# B&R Automation Studio project ControlPLC_DataDistribution (part 7)

#### vfValveBasic.st
```iecst
FUNCTION_BLOCK vfValveBasic

	pCommandWriteBack ACCESS (Inputs.adrCommands);

	IF NOT (Inputs.parameters.enabled) THEN
		internal.valveState	:= vfVALVE_BASIC_STOP;
	ELSIF(Inputs.commands.stop = TRUE) THEN
		pCommandWriteBack.stop := FALSE;
		internal.valveState	:= vfVALVE_BASIC_STOP;
	END_IF

	CASE internal.valveState OF

		vfVALVE_BASIC_WAIT_FOR_COMMANDS:

			Outputs.status.fbState := 'WAITING FOR COMMANDS';

			Outputs.status.readyForCommand := TRUE;

			IF (Inputs.commands.cycle = TRUE) THEN

				pCommandWriteBack.cycle := FALSE;

				internal.valveState	:= vfVALVE_BASIC_CYCLE_OPEN;

			ELSIF (Inputs.commands.open = TRUE) THEN

				pCommandWriteBack.open := FALSE;

				IF NOT Outputs.status.opened THEN

					internal.valveTimeOutTimer.IN := TRUE;

					internal.valveState	:= vfVALVE_BASIC_OPEN;
				END_IF

			ELSIF (Inputs.commands.close = TRUE)THEN

				pCommandWriteBack.close := FALSE;

				IF NOT Outputs.status.closed THEN

					internal.valveTimeOutTimer.IN := TRUE;

					internal.valveState	:= vfVALVE_BASIC_CLOSE;;
				END_IF

			END_IF

		vfVALVE_BASIC_CYCLE_OPEN:

			Outputs.status.fbState := 'CYCLE OPEN';
			Outputs.OpenValveSignal := TRUE; //cmd
			Outputs.CloseValveSignal := FALSE;//cmd
			Outputs.status.cycling	:= TRUE;//status
			Outputs.status.doOpen 	:= TRUE;//status
			Outputs.status.doClose	:= FALSE;//status

			internal.valveCycleTimer.PT	:= Inputs.parameters.cycleTime;
			internal.valveCycleTimer.IN	:= TRUE;
			internal.valveTimeOutTimer.IN := TRUE;

			//once its opened stop monitoring for timeout error
			IF Outputs.status.opened THEN
				internal.valveTimeOutTimer.IN := FALSE;

			//didnt open after allowed time
			ELSIF internal.valveTimeOutTimer.Q 	THEN
				internal.valveTimeOutTimer.IN := FALSE;
				internal.valveState := vfVALVE_BASIC_ERROR;

			END_IF

			//cycled open long enough
			IF (internal.valveCycleTimer.Q = TRUE) AND Outputs.status.opened THEN
				internal.valveCycleTimer.IN	:= FALSE;
				Outputs.CloseValveSignal := TRUE;
				Outputs.OpenValveSignal := FALSE;
				Outputs.status.doOpen := FALSE;
				Outputs.status.doClose := TRUE;

				//reset timeout timer
				internal.valveTimeOutTimer.IN := FALSE;
				internal.valveState				:= vfVALVE_BASIC_CYCLE_CLOSE;

			END_IF

		vfVALVE_BASIC_CYCLE_CLOSE:

			Outputs.status.fbState := 'CYCLE CLOSE';

			IF Outputs.status.closed THEN
				Outputs.status.cycling := FALSE;
				internal.valveTimeOutTimer.IN := FALSE;
				internal.valveState				:= vfVALVE_BASIC_WAIT_FOR_COMMANDS;

			ELSIF internal.valveTimeOutTimer.Q THEN
				internal.valveTimeOutTimer.IN := FALSE;
				internal.valveState := vfVALVE_BASIC_ERROR;

			END_IF

		vfVALVE_BASIC_OPEN:

			Outputs.status.fbState := 'OPENING';

			//open valve
			Outputs.OpenValveSignal := TRUE;
			Outputs.CloseValveSignal := FALSE;

			//update valve output status
			Outputs.status.doOpen 					:= TRUE;
			Outputs.status.doClose					:= FALSE;

			IF Outputs.status.opened THEN

				//reset timeout timer
				internal.valveTimeOutTimer.IN := FALSE;
				internal.valveState				:= vfVALVE_BASIC_WAIT_FOR_COMMANDS;

			ELSIF internal.valveTimeOutTimer.Q 	THEN

				internal.valveState := vfVALVE_BASIC_ERROR;

			END_IF

		vfVALVE_BASIC_CLOSE:

			Outputs.status.fbState := 'CLOSING';

			Outputs.OpenValveSignal := FALSE;
			Outputs.CloseValveSignal := TRUE;

			//update valve output status
			Outputs.status.doOpen 					:= FALSE;
			Outputs.status.doClose 				:= TRUE;

			IF Outputs.status.closed THEN

				//reset timeout timer
				internal.valveTimeOutTimer.IN := FALSE;
				internal.valveState				:= vfVALVE_BASIC_WAIT_FOR_COMMANDS;

			ELSIF internal.valveTimeOutTimer.Q 	THEN

				internal.valveState := vfVALVE_BASIC_ERROR;

			END_IF

		vfVALVE_BASIC_STOP:

			Outputs.status.fbState := 'STOPPING';

			Outputs.OpenValveSignal := FALSE;
			Outputs.CloseValveSignal := FALSE;

			//reset timeout timer
			internal.valveTimeOutTimer.IN := FALSE;
			internal.valveCycleTimer.IN		:= FALSE;

			//update valve output status
			Outputs.status.cycling					:= FALSE;
			Outputs.status.doOpen 					:= FALSE;
			Outputs.status.doClose 				:= FALSE;
			internal.valveState				:= vfVALVE_BASIC_WAIT_FOR_COMMANDS;

		vfVALVE_BASIC_ERROR:

			Outputs.status.fbState := 'ERRORED';

			//reset timeout timer
			internal.valveTimeOutTimer.IN := FALSE;

			Outputs.status.error := TRUE;

			IF Inputs.commands.errReset THEN

				Outputs.status.error := FALSE;

				internal.valveState				:= vfVALVE_BASIC_WAIT_FOR_COMMANDS;
			END_IF

	END_CASE

	IF (internal.valveState = vfVALVE_BASIC_ERROR) OR (internal.valveState = vfVALVE_BASIC_WAIT_FOR_COMMANDS) THEN
		Outputs.status.busy := FALSE;
	ELSE
		Outputs.status.busy := TRUE;
	END_IF

	//so nothing gets queued and stuck
	IF internal.valveState <> vfVALVE_BASIC_WAIT_FOR_COMMANDS THEN

		Outputs.status.readyForCommand := FALSE;

		pCommandWriteBack.close := FALSE;
		pCommandWriteBack.open := FALSE;
		pCommandWriteBack.cycle := FALSE;

	END_IF

	IF Inputs.commands.errReset THEN
		Outputs.status.error := FALSE;
	END_IF

	//feedback for position
	IF Inputs.parameters.hasLimitSensors THEN

		Outputs.status.closed := Inputs.closeLimitSensor;
		Outputs.status.opened := Inputs.openLimitSensor;

		Outputs.status.middle := NOT(Inputs.closeLimitSensor OR Inputs.openLimitSensor);

		internal.valveTimeOutTimer.PT := Inputs.parameters.TimeOutValue;
		internal.valveTimeOutTimer();

	ELSE

		internal.actuationDelayTimer.PT := Inputs.parameters.actuationDelay;

		IF Outputs.status.doClose AND NOT internal.oldDoClose THEN
			Outputs.status.opened := FALSE;
			internal.actuationDelayTimer.IN := TRUE;

		ELSIF Outputs.status.doOpen AND NOT internal.oldDoOpen THEN
			Outputs.status.closed := FALSE;
			internal.actuationDelayTimer.IN := TRUE;
		END_IF

		IF internal.actuationDelayTimer.Q THEN
			internal.actuationDelayTimer.IN := FALSE;
			Outputs.status.closed := Outputs.status.doClose;
			Outputs.status.opened := Outputs.status.doOpen;
		END_IF

		internal.actuationDelayTimer();

		//for rising edge
		internal.oldDoOpen := Outputs.status.doOpen;
		internal.oldDoClose := Outputs.status.doClose;

	END_IF

	//init timer for cycle option
	internal.valveCycleTimer();

END_FUNCTION_BLOCK
```

- vfValveBasic_readMe.docx (binary file, 312023 bytes)
### Library Logical/Libraries/VF/VF_PARSER (IEC, version 1.00.0)

#### RevisionNotes.txt
```
****************************************************************************************************
IMPORTANT: Always update the library version number in the library Properties 'Details' tab.
****************************************************************************************************

Version 1.00 - 9/23/19, W. Stebler
----------------------------------
- Original version.
```

#### Types.typ - Exported data types
```iecst
(**)
(*ParseLSF structures*)

TYPE
	vfpLSFCommandType : 	STRUCT
		SelectedBuildLayout : UDINT;
		SelectedPrintNumber : UINT;
		SelectedRack : USINT;
		SelectedLayer : UDINT;
		OptionalStartingTrajectory : UINT;
		NumLasersInRack : USINT;
		OpenLayer : BOOL;
		ParseTrajectory : BOOL;
		CloseLayer : BOOL;
		AbortLayer : BOOL;
		ResetError : BOOL;
	END_STRUCT;
	vfpLSFStatusType : 	STRUCT
		LayerFilename : STRING[255];
		LayerOpen : BOOL;
		CurrentLayer : UDINT;
		FinalTrajectoryNumber : UINT;
		ParsedTrajectoryNumber : UINT;
		ParseTrajectoryComplete : BOOL;
		LayerClosed : BOOL;
		LayerAborted : BOOL;
		Error : BOOL;
		ErrorID : UINT;
		ErrorText : STRING[80];
	END_STRUCT;
	vfpLSFInternalFBType : 	STRUCT
		FileOpen : FileOpen;
		FileReadEx : FileReadEx;
		FileClose : FileClose;
	END_STRUCT;
	vfpLSFParsedDataType : 	STRUCT
		TrajectoryCircularBuffer : ARRAY[1..vfp_LSF_TRAJECTORY_FIFO_SIZE]OF vfpLSFBufferElementType;
		FIFOCount : USINT := 0;
		FIFOHeadIndex : USINT := 1;
		FIFOTailIndex : USINT := 1;
	END_STRUCT;
	vfpLSFBufferElementType : 	STRUCT
		TrajectoryNumber : UINT;
		LaserTrajectoryInfo : ARRAY[1..vfp_LSF_NUM_LASERS_PER_SYSTEM]OF vfpLSFLaserTrajectoryInfoType;
		ExitCode : UINT;
	END_STRUCT;
	vfpLSFLaserTrajectoryInfoType : 	STRUCT
		PowerSetpointPercent : REAL;
		NumStateValues : UINT;
		StateValue32Bit : ARRAY[1..vfp_LSF_MAX_32BIT_VAL_PER_TRAJ]OF UDINT;
	END_STRUCT;
	vfpLSFLocalType : 	STRUCT
		Step : vfpLSFStepsEnum;
		StepTrace : ARRAY[0..99]OF vfpLSFStepsEnum;
		index : UINT;
		FB : vfpLSFInternalFBType;
		ErrorStep : vfpLSFStepsEnum;
		DataBuffer : STRING[vfp_LSF_FILE_READ_BUFFER_SIZE];
		ReadLengthBytes : UDINT;
		TotalBytesRead : UDINT;
		StartingByteAddress : UDINT;
		MaxBytes : UDINT;
		NextByteAddress : UDINT;
		CurrentByteIndex : UDINT;
		ParameterValue : LREAL;
		ParameterValue_UDINT : UDINT;
		ParameterValue_string : STRING[vfp_MAX_CHARS_PER_STRING_VALUE];
		ParsedHeaderLine : BOOL;
		FoundTrajectory : BOOL;
		Status : UINT;
		BuildLayout : UDINT;
		PrintNumber : UINT;
		RackNumber : USINT;
		LayerNumber : UDINT;
		LayerClosed : BOOL;
		LayerAborted : BOOL;
		FinalTrajectoryNumber : UINT;
		TrajectoryNumber : UINT;
		LaserNumber : USINT;
		LastLaserNumber : USINT;
		LaserPowerValueIndex : USINT;
		LaserStateValueIndex : UINT;
		ExpectedNumEvents : UINT;
		FileReadOffset : UDINT;
		LocalFileHandle : UDINT;
		GCodeLineNumber_string : STRING[30];
		BuildLayout_string : STRING[20];
		PrintNumber_string : STRING[20];
		RackNumber_string : STRING[8];
		LayerNumber_string : STRING[8];
		LayerFileName : STRING[255];
		HeaderElement : USINT;
		BuildName : STRING[80];
		BuildPlateFormat : STRING[40];
		Temp_val : UINT;
		Temp_string : STRING[40];
	END_STRUCT;
	vfpLSFStepsEnum :
		(
		vfSTEP_LSF_INITIALIZE,
		vfSTEP_LSF_IDLE,
		vfSTEP_LSF_CREATE_LAYER_FILENAME,
		vfSTEP_LSF_OPEN_FILE,
		vfSTEP_LSF_WAIT_FILE_OPEN,
		vfSTEP_LSF_AWAIT_COMMAND,
		vfSTEP_LSF_READ_FILE_DATA,
		vfSTEP_LSF_WAIT_READ_DONE,
		vfSTEP_LSF_PARSE_FILE_HDR,
		vfSTEP_LSF_FIND_TRAJECTORY_HDR,
		vfSTEP_LSF_PARSE_TRAJECTORY_HDR,
		vfSTEP_LSF_PARSE_NUM_EVENTS,
		vfSTEP_LSF_PARSE_LASER_POWERS,
		vfSTEP_LSF_PARSE_LASER_STATES,
		vfSTEP_LSF_SELECT_NEXT_LASER,
		vfSTEP_LSF_TRAJECTORY_PARSE_DONE,
		vfSTEP_LSF_AWAIT_NEXT_COMMAND,
		vfSTEP_LSF_CLOSE_FILE,
		vfSTEP_LSF_WAIT_FILE_CLOSED,
		vfSTEP_LSF_LAYER_CLOSED,
		vfSTEP_LSF_LAYER_ABORTED,
		vfSTEP_LSF_ERROR,
		vfSTEP_LSF_AWAIT_CMD_RESET
		);
END_TYPE

(**)
(*ParseFEF structures*)

TYPE
	vfpFEFCommandType : 	STRUCT
		SelectedBuildLayout : UDINT;
		SelectedPrintNumber : UINT;
		SelectedLayer : UDINT;
		OptionalStartingTrajectory : UINT;
		OpenLayer : BOOL;
		ParseTrajectory : BOOL;
		CloseLayer : BOOL;
		AbortLayer : BOOL;
		ResetError : BOOL;
	END_STRUCT;
	vfpFEFStatusType : 	STRUCT
		LayerFilename_GCode : STRING[255];
		LayerFilename_FixedEvents : STRING[255];
		LayerOpen : BOOL;
		CurrentLayer : UDINT;
		FinalTrajectoryNumber : UINT;
		ParsedTrajectoryNumber : UINT;
		ParseTrajectoryComplete : BOOL;
		LayerClosed : BOOL;
		LayerAborted : BOOL;
		Error : BOOL;
		ErrorID : UINT;
		ErrorText : STRING[80];
	END_STRUCT;
	vfpFEFInternalFBType : 	STRUCT
		FileOpen : FileOpen;
		FileReadEx : FileReadEx;
		FileClose : FileClose;
	END_STRUCT;
	vfpFEFParsedDataType : 	STRUCT
		TrajectoryCircularBuffer : ARRAY[1..vfp_FEF_TRAJECTORY_FIFO_SIZE]OF vfpFEFBufferElementType;
		FIFOCount : USINT := 0;
		FIFOHeadIndex : USINT := 1;
		FIFOTailIndex : USINT := 1;
	END_STRUCT;
	vfpFEFBufferElementType : 	STRUCT
		TrajectoryNumber : UINT;
		ExitCode : UINT;
		MasterAxis : USINT;
		StartPositionMM : REAL;
		EndPositionMM : REAL;
		EventPeriodMM : REAL;
	END_STRUCT;
	vfpFEFLocalType : 	STRUCT
		Step : vfpFEFStepsEnum;
		StepTrace : ARRAY[0..99]OF vfpFEFStepsEnum;
		index : UINT;
		FB : vfpFEFInternalFBType;
		ErrorStep : vfpFEFStepsEnum;
		DataBuffer : STRING[vfp_FEF_FILE_READ_BUFFER_SIZE];
		ReadLengthBytes : UDINT;
		TotalBytesRead : UDINT;
		StartingByteAddress : UDINT;
		MaxBytes : UDINT;
		NextByteAddress : UDINT;
		CurrentByteIndex : UDINT;
		ParameterValue : LREAL;
		ParameterValue_UDINT : UDINT;
		ParameterValue_string : STRING[vfp_MAX_CHARS_PER_STRING_VALUE];
		ParsedHeaderLine : BOOL;
		FoundTrajectory : BOOL;
		Status : UINT;
		BuildLayout : UDINT;
		PrintNumber : UINT;
		LayerNumber : UDINT;
		LayerClosed : BOOL;
		LayerAborted : BOOL;
		FinalTrajectoryNumber : UINT;
		TrajectoryNumber : UINT;
		FileReadOffset : UDINT;
		LocalFileHandle : UDINT;
		MasterAxis : USINT;
		StartPosition : REAL;
		EndPosition : REAL;
		EventPeriod : REAL;
		GCodeLineNumber_string : STRING[30];
		BuildLayout_string : STRING[20];
		PrintNumber_string : STRING[20];
		LayerNumber_string : STRING[8];
		LayerFileName_FixedEvents : STRING[255];
		LayerFileName_GCode : STRING[255];
		HeaderElement : USINT;
		BuildName : STRING[80];
		BuildPlateFormat : STRING[40];
		Temp_val : UINT;
		Temp_string : STRING[40];
	END_STRUCT;
	vfpFEFStepsEnum :
		(
		vfSTEP_FEF_INITIALIZE,
		vfSTEP_FEF_IDLE,
		vfSTEP_FEF_CREATE_LAYER_FILENAME,
		vfSTEP_FEF_OPEN_FILE,
		vfSTEP_FEF_WAIT_FILE_OPEN,
		vfSTEP_FEF_AWAIT_COMMAND,
		vfSTEP_FEF_READ_FILE_DATA,
		vfSTEP_FEF_WAIT_READ_DONE,
		vfSTEP_FEF_PARSE_FILE_HDR,
		vfSTEP_FEF_FIND_TRAJECTORY_HDR,
		vfSTEP_FEF_PARSE_TRAJECTORY_HDR,
		vfSTEP_FEF_PARSE_MASTER_AXIS,
		vfSTEP_FEF_PARSE_START_POSN,
		vfSTEP_FEF_PARSE_END_POSN,
		vfSTEP_FEF_PARSE_EVENT_PERIOD,
		vfSTEP_FEF_TRAJECTORY_PARSE_DONE,
		vfSTEP_FEF_AWAIT_NEXT_COMMAND,
		vfSTEP_FEF_CLOSE_FILE,
		vfSTEP_FEF_WAIT_FILE_CLOSED,
		vfSTEP_FEF_LAYER_CLOSED,
		vfSTEP_FEF_LAYER_ABORTED,
		vfSTEP_FEF_ERROR,
		vfSTEP_FEF_AWAIT_CMD_RESET
		);
END_TYPE

(**)
(*SMRFile structures*)

TYPE
	VfSMRFileInternalType : 	STRUCT
		Step : VfSMRFileStepsEnum;
		StepTrace : ARRAY[0..99]OF VfSMRFileStepsEnum;
		ErrorStep : VfSMRFileStepsEnum;
		FB : VfSMRFileInternalFBType;
		index : UINT;
	END_STRUCT;
	VfSMRFileInternalFBType : 	STRUCT
		FileCopy1 : FileCopy;
		FileCopy2 : FileCopy;
		FileCopy3 : FileCopy;
	END_STRUCT;
	VfSMRFileStepsEnum :
		(
		vfSMR_FILE_STEP_IDLE,
		vfSMR_FILE_STEP_COPY_TO_SMR1,
		vfSMR_FILE_STEP_COPY_TO_SMR2,
		vfSMR_FILE_STEP_COPY_TO_SMR3,
		vfSMR_FILE_STEP_COPY_TO_SMR4,
		vfSMR_FILE_STEP_COPY_TO_PTR1,
		vfSMR_FILE_STEP_COPY_TO_PTR2,
		vfSMR_FILE_STEP_COPY_TO_LCR1,
		vfSMR_FILE_STEP_COPY_TO_LCR2,
		vfSMR_FILE_STEP_DONE,
		vfSMR_FILE_STEP_DISCONNECT1,
		vfSMR_FILE_STEP_DISCONNECT2,
		vfSMR_FILE_STEP_ERROR,
		vfSMR_FILE_STEP_ERROR_RESET
		);
END_TYPE

(**)
(*SMRConnect structures*)

TYPE
	VfSMRConnectInternalType : 	STRUCT
		Step : VfSMRConnectStepsEnum;
		StepTrace : ARRAY[0..99]OF VfSMRConnectStepsEnum;
		ErrorStep : VfSMRConnectStepsEnum;
		FB : VfSMRConnectInternalFBType;
		LocalFileHandle : UDINT;
		index : UINT;
	END_STRUCT;
	VfSMRConnectInternalFBType : 	STRUCT
		DevLinkRemote : DevLink;
		DevLinkLocalSMR : DevLink;
		DevLinkLocalPTR : DevLink;
		DevLinkLocalLCR : DevLink;
		DevUnlinkRemote : DevUnlink;
		DevUnlinkLocalSMR : DevUnlink;
		DevUnlinkLocalPTR : DevUnlink;
		DevUnlinkLocalLCR : DevUnlink;
	END_STRUCT;
	VfSMRConnectStepsEnum :
		(
		vfSMR_CNCT_STEP_IDLE,
		vfSMR_CNCT_STEP_CONNECT_SMR1,
		vfSMR_CNCT_STEP_CONNECT_SMR2,
		vfSMR_CNCT_STEP_CONNECT_PTR1,
		vfSMR_CNCT_STEP_CONNECT_PTR2,
		vfSMR_CNCT_STEP_CONNECT_LCR1,
		vfSMR_CNCT_STEP_CONNECT_LCR2,
		vfSMR_CNCT_STEP_CONNECT_REMOTE1,
		vfSMR_CNCT_STEP_CONNECT_REMOTE2,
		vfSMR_CNCT_STEP_DONE,
		vfSMR_CNCT_STEP_DISCONNECT1,
		vfSMR_CNCT_STEP_DISCONNECT2,
		vfSMR_CNCT_STEP_ERROR,
		vfSMR_CNCT_STEP_ERROR_RESET
		);
END_TYPE

(**)
(*LCRConnect structures*)

TYPE
	VfLCRConnectInternalType : 	STRUCT
		Step : VfLCRConnectStepsEnum;
		StepTrace : ARRAY[0..99]OF VfLCRConnectStepsEnum;
		ErrorStep : VfLCRConnectStepsEnum;
		FB : VfLCRConnectInternalFBType;
		LocalFileName : STRING[80];
		LocalLCRDriveName : STRING[80];
		LocalFileHandle : UDINT;
		i : UINT;
	END_STRUCT;
	VfLCRConnectInternalFBType : 	STRUCT
		DevLinkLocalLCR : DevLink;
		DevUnlinkLocalLCR : DevUnlink;
	END_STRUCT;
	VfLCRConnectStepsEnum :
		(
		vfLCR_CNCT_STEP_IDLE,
		vfLCR_CNCT_STEP_CONNECT_LCR1,
		vfLCR_CNCT_STEP_CONNECT_LCR2,
		vfLCR_CNCT_STEP_DONE,
		vfLCR_CNCT_STEP_DISCONNECT1,
		vfLCR_CNCT_STEP_DISCONNECT2,
		vfLCR_CNCT_STEP_ERROR,
		vfLCR_CNCT_STEP_ERROR_RESET
		);
END_TYPE
```

#### Constants.var - Exported constants
```iecst
(*Shared parser constants*)
VAR CONSTANT
	vfp_MAX_CHARS_PER_STRING_VALUE : UINT := 60; (*Maximum characters allowed for any string value*)
	vfp_MAX_CHARS_PER_NUMERIC_VALUE : UINT := 30; (*Maximum characters allowed for any numeric value (including decimal point, negative sign, delimiter)*)
	fvp_FIRST_TRAJECTORY_NUMBER : UINT := 10; (*Trajectories start at N0010 and increment by 10 (N0010, N0020, N0030,...)*)
	fvp_TRAJECTORY_NUMBER_INCREMENT : USINT := 10;
END_VAR
(*Laser State File (LSF) parser constants*)
VAR CONSTANT
	vfp_LSF_FILE_READ_BUFFER_SIZE : UDINT := 341000; (*> maximum single trajectory (1630 values * 11 bytes * 19 lasers)*)
	vfp_LSF_TRAJECTORY_FIFO_SIZE : USINT := 4;
	vfp_LSF_NUM_LASERS_PER_SYSTEM : UINT := 19;
	vfp_LSF_MAX_32BIT_VAL_PER_TRAJ : UINT := 1630; (*52000 events / 32 bits = 1625 (+ 5 extra for padding)*)
	vfp_LSF_MAX_CHARS_PER_32BIT_VAL : UINT := 11; (*Maximum characters allowed for a laser state event (10 digit value + delimiter) [10 digits required to represent max UDINT value of 4,294,967,295]*)
	vfp_LSF_MAX_CHARS_PER_HEADER : UINT := 300; (*Maximum characters allowed for a single trajectory header information*)
END_VAR
(*Fixed Event File (FEF) parser constants*)
VAR CONSTANT
	vfp_FEF_FILE_READ_BUFFER_SIZE : UDINT := 200;
	vfp_FEF_TRAJECTORY_FIFO_SIZE : USINT := 100;
	vfp_FEF_MASTER_AXIS_X : USINT := 1;
	vfp_FEF_MASTER_AXIS_Y : USINT := 2;
	vfp_FEF_MAX_X_Y_POSN_MM : LREAL := 960.0;
END_VAR
(*Common parser ASCII character codes*)
VAR CONSTANT
	vfp_CHAR_CARRIAGE_RETURN : USINT := 13; (*Carriage Return ASCII char*)
	vfp_CHAR_LINE_FEED : USINT := 10; (*Line Feed ASCII char*)
	vfp_CHAR_SPACE : USINT := 32; (*Space ASCII char*)
	vfp_CHAR_COMMA : USINT := 44; (*',' ASCII char*)
	vfp_CHAR_DECIMAL_POINT : USINT := 46; (*'.' ASCII char*)
	vfp_CHAR_DIGIT_0 : USINT := 48; (*'0' ASCII char*)
	vfp_CHAR_DIGIT_9 : USINT := 57; (*'9' ASCII char*)
	vfp_CHAR_EQUALS : USINT := 61; (*'=' ASCII char*)
	vfp_CHAR_TRAJECTORY_HDR : USINT := 78; (*'N' ASCII char*)
END_VAR
(*Common parser return codes*)
VAR CONSTANT
	vfp_ERR_OK : UINT := 50000;
	vfp_ERR_EOL_REACHED : UINT := 50001;
	vfp_ERR_NO_MORE_LINES : UINT := 50002;
	vfp_ERR_NULL_POINTER : UINT := 50003;
	vfp_ERR_INVALID_PARAMETER : UINT := 50004;
	vfp_ERR_NO_DELIMITER : UINT := 50005;
	vfp_ERR_MISSING_DATA : UINT := 50006;
	vfp_ERR_NON_NUMERICAL : UINT := 50007;
	vfp_ERR_WRONG_NUM_STATES : UINT := 50008;
	vfp_ERR_BAD_HEADER : UINT := 50009;
	vfp_ERR_HEADER_INVALID_NUM_TRAJ : UINT := 50010;
	vfp_ERR_BUFFER_SIZE : UINT := 50040;
	vfp_ERR_FATAL_SYSTEM_ERROR : UINT := 50050;
END_VAR
(**)
```

#### VF_PARSER.fun - Exported functions and function blocks
```iecst
{REDUND_ERROR} FUNCTION GetNextString : UINT (* *) (*$GROUP=User,$CAT=User,$GROUPICON=User.png,$CATICON=User.png*)
	VAR_INPUT
		pAdrData : UDINT;
		pParameter : UDINT;
	END_VAR
	VAR
		AdrData : REFERENCE TO UDINT;
		CharVal : REFERENCE TO USINT;
		index : UINT;
		ParameterValue : REFERENCE TO STRING[vfp_MAX_CHARS_PER_STRING_VALUE];
		TempString : STRING[vfp_MAX_CHARS_PER_STRING_VALUE];
	END_VAR
END_FUNCTION

{REDUND_ERROR} FUNCTION GetNextParameter : UINT (* *) (*$GROUP=User,$CAT=User,$GROUPICON=User.png,$CATICON=User.png*)
	VAR_INPUT
		pAdrData : UDINT;
		pParameter : UDINT;
	END_VAR
	VAR
		AdrData : REFERENCE TO UDINT;
		CharVal : REFERENCE TO USINT;
		index : UINT;
		ParameterValue : REFERENCE TO LREAL;
		TempString : STRING[vfp_MAX_CHARS_PER_NUMERIC_VALUE];
	END_VAR
END_FUNCTION

{REDUND_ERROR} FUNCTION FindNextLineStart : UINT (* *) (*$GROUP=User,$CAT=User,$GROUPICON=User.png,$CATICON=User.png*)
	VAR_INPUT
		pAdrData : UDINT;
		MaxBytes : UDINT;
	END_VAR
	VAR
		AdrData : REFERENCE TO UDINT;
		CharVal : REFERENCE TO USINT;
		index : UDINT;
	END_VAR
END_FUNCTION

{REDUND_ERROR} FUNCTION FindNextTrajectoryStart : UINT (* *) (*$GROUP=User,$CAT=User,$GROUPICON=User.png,$CATICON=User.png*)
	VAR_INPUT
		pAdrData : UDINT;
		MaxBytes : UDINT;
	END_VAR
	VAR
		AdrData : REFERENCE TO UDINT;
		CharVal : REFERENCE TO USINT;
		index : UDINT;
	END_VAR
END_FUNCTION

{REDUND_ERROR} FUNCTION GetSystemErrorText : BOOL (* *) (*$GROUP=User,$CAT=User,$GROUPICON=User.png,$CATICON=User.png*)
	VAR_INPUT
		ErrorID : UINT;
		ErrorText : REFERENCE TO STRING[80];
	END_VAR
END_FUNCTION

{REDUND_ERROR} {REDUND_UNREPLICABLE} FUNCTION_BLOCK VfSMRFileSetup (*Not currently in use*) (*$GROUP=User,$CAT=User,$GROUPICON=User.png,$CATICON=User.png*)
	VAR_INPUT
		Execute : {REDUND_UNREPLICABLE} BOOL;
		ErrorReset : {REDUND_UNREPLICABLE} BOOL;
		pPEFName : {REDUND_UNREPLICABLE} UDINT;
		pFEFName : {REDUND_UNREPLICABLE} UDINT;
		pRemoteDriveName : {REDUND_UNREPLICABLE} UDINT;
		pLocalSMRDriveName : {REDUND_UNREPLICABLE} UDINT;
		pLocalPTRDriveName : {REDUND_UNREPLICABLE} UDINT;
		pLocalLCRDriveName : {REDUND_UNREPLICABLE} UDINT;
	END_VAR
	VAR_OUTPUT
		Done : {REDUND_UNREPLICABLE} BOOL;
		Error : {REDUND_UNREPLICABLE} BOOL;
		ErrorID : {REDUND_UNREPLICABLE} UINT;
	END_VAR
	VAR
		Internal : {REDUND_UNREPLICABLE} VfSMRFileInternalType;
	END_VAR
END_FUNCTION_BLOCK

{REDUND_UNREPLICABLE} FUNCTION_BLOCK VfSMRConnect (*Not currently in use*)
	VAR_INPUT
		Execute : {REDUND_UNREPLICABLE} BOOL;
		ErrorReset : {REDUND_UNREPLICABLE} BOOL;
		pRemoteDriveName : {REDUND_UNREPLICABLE} UDINT;
		pLocalSMRDriveName : {REDUND_UNREPLICABLE} UDINT;
		pLocalPTRDriveName : {REDUND_UNREPLICABLE} UDINT;
		pLocalLCRDriveName : {REDUND_UNREPLICABLE} UDINT;
		pRemoteDrive : {REDUND_UNREPLICABLE} UDINT;
		pLocalSMRDrive : {REDUND_UNREPLICABLE} UDINT;
		pLocalPTRDrive : {REDUND_UNREPLICABLE} UDINT;
		pLocalLCRDrive : {REDUND_UNREPLICABLE} UDINT;
	END_VAR
	VAR_OUTPUT
		Done : {REDUND_UNREPLICABLE} BOOL;
		Error : {REDUND_UNREPLICABLE} BOOL;
		ErrorID : {REDUND_UNREPLICABLE} UINT;
		LocalSMRDriveHandle : {REDUND_UNREPLICABLE} UDINT;
		LocalPTRDriveHandle : {REDUND_UNREPLICABLE} UDINT;
		LocalLCRDriveHandle : {REDUND_UNREPLICABLE} UDINT;
		RemoteDriveHandle : {REDUND_UNREPLICABLE} UDINT;
	END_VAR
	VAR
		Internal : {REDUND_UNREPLICABLE} VfSMRConnectInternalType;
	END_VAR
END_FUNCTION_BLOCK

{REDUND_ERROR} {REDUND_UNREPLICABLE} FUNCTION_BLOCK VfLCRConnect (*Not currently in use*) (*$GROUP=User,$CAT=User,$GROUPICON=User.png,$CATICON=User.png*)
	VAR_INPUT
		Execute : {REDUND_UNREPLICABLE} BOOL;
		ErrorReset : {REDUND_UNREPLICABLE} BOOL;
		pLocalLCRDriveName : {REDUND_UNREPLICABLE} UDINT;
		pLocalLCRDrive : {REDUND_UNREPLICABLE} UDINT;
	END_VAR
	VAR_OUTPUT
		Done : {REDUND_UNREPLICABLE} BOOL;
		Error : {REDUND_UNREPLICABLE} BOOL;
		ErrorID : {REDUND_UNREPLICABLE} UINT;
		LocalLCRDriveHandle : {REDUND_UNREPLICABLE} UDINT;
	END_VAR
	VAR
		Internal : {REDUND_UNREPLICABLE} VfLCRConnectInternalType;
	END_VAR
END_FUNCTION_BLOCK

{REDUND_ERROR} {REDUND_UNREPLICABLE} FUNCTION_BLOCK VfParseLaserStateFile (* *) (*$GROUP=User,$CAT=User,$GROUPICON=User.png,$CATICON=User.png*)
	VAR_INPUT
		Enable : {REDUND_UNREPLICABLE} BOOL;
		pParsedData : REFERENCE TO vfpLSFParsedDataType;
		Command : {REDUND_UNREPLICABLE} vfpLSFCommandType;
	END_VAR
	VAR_OUTPUT
		Active : {REDUND_UNREPLICABLE} BOOL;
		Status : {REDUND_UNREPLICABLE} vfpLSFStatusType;
	END_VAR
	VAR
		local : {REDUND_UNREPLICABLE} vfpLSFLocalType;
	END_VAR
END_FUNCTION_BLOCK

{REDUND_ERROR} {REDUND_UNREPLICABLE} FUNCTION_BLOCK VfParseFixedEventFile (* *) (*$GROUP=User,$CAT=User,$GROUPICON=User.png,$CATICON=User.png*)
	VAR_INPUT
		Enable : {REDUND_UNREPLICABLE} BOOL;
		pParsedData : REFERENCE TO vfpFEFParsedDataType;
		Command : {REDUND_UNREPLICABLE} vfpFEFCommandType;
	END_VAR
	VAR_OUTPUT
		Active : {REDUND_UNREPLICABLE} BOOL;
		Status : {REDUND_UNREPLICABLE} vfpFEFStatusType;
	END_VAR
	VAR
		local : {REDUND_UNREPLICABLE} vfpFEFLocalType;
	END_VAR
END_FUNCTION_BLOCK
```

#### VfParseLaserStateFile.st - Laser state file parser
```iecst
// Laser State File format:
//
//	BuildName, Layer, TotalLayers, TotalTrajectories, BuildPlateFormat, RackNumber
//	N0010,NumEvents,Laser1Power,Laser2Power,Laser3Power,…Laser19Power
//	Laser1LSW1,Laser1LSW2,Laser1LSW3,…Laser1LSW<NumEvents>
//	Laser2LSW1,Laser2LSW2,Laser2LSW3,…Laser2LSW<NumEvents>
//	Laser3LSW1,Laser3LSW2,Laser3LSW3,…Laser3LSW<NumEvents>
//	…
//	Laser19LSW1,Laser19LSW2,Laser19LSW3,…Laser19LSW<NumEvents>
//	N0020,NumEvents,Laser1Power,Laser2Power,Laser3Power,…Laser19Power
//	Laser1LSW1,Laser1LSW2,Laser1LSW3,…Laser1LSW<NumEvents>
//	Laser2LSW1,Laser2LSW2,Laser2LSW3,…Laser2LSW<NumEvents>
//
//
//	BuildName = Name of the build being processed (string)
//	Layer = Current layer number (int)
//	TotalLayers = Total number of layers (int)
//	TotalTrajectories = Total number of trajectories on current layer (int)
//	BuildPlateFormat = build plate format used, [200x600, 400x600, 600x600] (string)
//	RackNumber = The rack for the current file (int) [1..8]
//
//	Nxxxx = print trajectory number; will always start at 0010 and increment by 10; always 4 digits
//	NumEvents = the number of events in that trajectory (can be used as an error check)
//	LaserNPower = the % power value for LaserN during that trajectory move

FUNCTION_BLOCK VfParseLaserStateFile

	IF (Enable) THEN

		// Trace the currently-active step; the most recent step is in array index [0].
		IF (local.Step <> local.StepTrace[0]) THEN
			// Use the line below to determined the number of scans required for each operation.
			// IF (local.Step <> vfSTEP_LSF_INITIALIZE) AND (local.Step <> vfSTEP_LSF_IDLE) AND (local.Step <> vfSTEP_LSF_AWAIT_NEXT_COMMAND) AND (local.Step <> vfSTEP_LSF_ERROR) AND (local.Step <> vfSTEP_LSF_AWAIT_CMD_RESET) THEN
			FOR local.index := 99 TO 1 BY (-1) DO
				local.StepTrace[local.index] := local.StepTrace[local.index-1];
			END_FOR
			local.StepTrace[0] := local.Step;
		END_IF

		CASE local.Step OF

			// ------------------------------------------------------------------------------------------------------------------------------------------------
			// Initialize parser state.
			vfSTEP_LSF_INITIALIZE:
				Status.LayerFilename := '';
				Status.LayerOpen := FALSE;
				Status.CurrentLayer := 0;
				Status.ParsedTrajectoryNumber := 0;
				Status.ParseTrajectoryComplete := FALSE;
				Status.LayerClosed := FALSE;
				Status.LayerAborted := FALSE;
				Status.Error := FALSE;
				Status.ErrorID := ERR_OK;

				local.FB.FileOpen.enable := FALSE;
				local.FB.FileReadEx.enable := FALSE;
				local.FB.FileClose.enable := FALSE;

				local.ParsedHeaderLine := FALSE;
				local.FoundTrajectory := FALSE;
				local.TrajectoryNumber := fvp_FIRST_TRAJECTORY_NUMBER;
				local.FinalTrajectoryNumber := 0;
				local.LayerAborted := FALSE;
				local.LayerClosed := FALSE;

				IF NOT (Command.ParseTrajectory OR Command.OpenLayer OR Command.CloseLayer OR Command.AbortLayer OR Command.ResetError) THEN
					local.Step := vfSTEP_LSF_IDLE;
				END_IF

				// ------------------------------------------------------------------------------------------------------------------------------------------------
				// Wait for incoming command to open the specified layer file.
			vfSTEP_LSF_IDLE:
				Active := TRUE;

				Status.LayerFilename := '';
				local.ParsedHeaderLine := FALSE;
				local.FoundTrajectory := FALSE;
				local.TrajectoryNumber := fvp_FIRST_TRAJECTORY_NUMBER;
				local.FinalTrajectoryNumber := 0;
				local.LayerAborted := FALSE;
				local.LayerClosed := FALSE;

				IF (Command.OpenLayer) AND NOT (Command.CloseLayer OR Command.AbortLayer OR Command.ResetError) THEN
					IF (Command.SelectedBuildLayout > 0) AND (Command.SelectedPrintNumber > 0) AND (Command.SelectedRack > 0) THEN
						local.BuildLayout := Command.SelectedBuildLayout;
						local.PrintNumber := Command.SelectedPrintNumber;
						local.RackNumber := Command.SelectedRack;
						local.LastLaserNumber := Command.NumLasersInRack;
						local.LayerNumber := Command.SelectedLayer;
						local.Step := vfSTEP_LSF_CREATE_LAYER_FILENAME;
					END_IF
				ELSIF (Command.AbortLayer) THEN
					local.LayerAborted := TRUE;
					local.Step := vfSTEP_LSF_CLOSE_FILE;
				END_IF

				// ------------------------------------------------------------------------------------------------------------------------------------------------
			vfSTEP_LSF_CREATE_LAYER_FILENAME:

				// Convert the desired build layout number to a string with the "XXXXX" format, adding required leading 0s.
				brsitoa(local.BuildLayout, ADR(local.Temp_string));
				IF (local.BuildLayout > 9999) THEN
					local.BuildLayout_string := '';
				ELSIF (local.BuildLayout > 999) THEN
					local.BuildLayout_string := '0';
				ELSIF (local.BuildLayout > 99) THEN
					local.BuildLayout_string := '00';
				ELSIF (local.BuildLayout > 9) THEN
					local.BuildLayout_string := '000';
				ELSE
					local.BuildLayout_string := '0000';
				END_IF
				brsstrcat(ADR(local.BuildLayout_string), ADR(local.Temp_string));

				// Convert the desired print number to a string with the "YYYY" format, adding required leading 0s.
				brsitoa(local.PrintNumber, ADR(local.Temp_string));
				IF (local.PrintNumber > 999) THEN
					local.PrintNumber_string := '';
				ELSIF (local.PrintNumber > 99) THEN
					local.PrintNumber_string := '0';
				ELSIF (local.PrintNumber > 9) THEN
					local.PrintNumber_string := '00';
				ELSE
					local.PrintNumber_string := '000';
				END_IF
				brsstrcat(ADR(local.PrintNumber_string), ADR(local.Temp_string));

				// Convert the desired layer number to a string with the "nnnnn" format, adding required leading 0s.
				brsitoa(local.LayerNumber, ADR(local.Temp_string));
				IF (local.LayerNumber > 9999) THEN
					 local.LayerNumber_string := '';
				ELSIF (local.LayerNumber > 999) THEN
					local.LayerNumber_string := '0';
				ELSIF (local.LayerNumber > 99) THEN
					local.LayerNumber_string := '00';
				ELSIF (local.LayerNumber > 9) THEN
					local.LayerNumber_string := '000';
				ELSE
					local.LayerNumber_string := '0000';
				END_IF
				brsstrcat(ADR(local.LayerNumber_string), ADR(local.Temp_string));

				// Convert the desired rack number to a string with the "rr" format, adding required leading 0s.
				brsitoa(local.RackNumber, ADR(local.Temp_string));
				IF (local.RackNumber > 9) THEN
					local.RackNumber_string := '';
				ELSE
					local.RackNumber_string := '0';
				END_IF
				brsstrcat(ADR(local.RackNumber_string), ADR(local.Temp_string));

				// Format the complete layer filename.
				// The .vflc file type extension stands for Vulcan Forms Laser Control
				local.LayerFileName := 'VF-';
				brsstrcat(ADR(local.LayerFileName), ADR(local.BuildLayout_string));
				brsstrcat(ADR(local.LayerFileName), ADR('-'));
				brsstrcat(ADR(local.LayerFileName), ADR(local.PrintNumber_string));
				brsstrcat(ADR(local.LayerFileName), ADR('_L'));
				brsstrcat(ADR(local.LayerFileName), ADR(local.LayerNumber_string));
				brsstrcat(ADR(local.LayerFileName), ADR('_LaserControl_R'));
				brsstrcat(ADR(local.LayerFileName), ADR(local.RackNumber_string));
				brsstrcat(ADR(local.LayerFileName), ADR('.vflc'));

				Status.LayerFilename := local.LayerFileName;
				local.Step := vfSTEP_LSF_OPEN_FILE;

				// ------------------------------------------------------------------------------------------------------------------------------------------------
				// Open the laser state file for the specified layer in read-only mode.
			vfSTEP_LSF_OPEN_FILE:
				local.FB.FileOpen.pDevice := ADR('CurrentLaserControlFiles');
				local.FB.FileOpen.pFile := ADR(local.LayerFileName);
				local.FB.FileOpen.mode := fiREAD_ONLY;
				local.FB.FileOpen.enable := TRUE;
				local.Step := vfSTEP_LSF_WAIT_FILE_OPEN;

				// ------------------------------------------------------------------------------------------------------------------------------------------------
				// Wait for file to be open or failure.
			vfSTEP_LSF_WAIT_FILE_OPEN:
				IF (local.FB.FileOpen.status = ERR_OK) THEN
					local.FB.FileOpen.enable := FALSE;
					local.LocalFileHandle := local.FB.FileOpen.ident;
					local.FileReadOffset := 0;
					// Notify the caller that the requested layer is open.
					Status.LayerOpen := TRUE;
					Status.CurrentLayer := local.LayerNumber;
					local.Step := vfSTEP_LSF_AWAIT_COMMAND;

				ELSIF (local.FB.FileOpen.status <> ERR_FUB_BUSY) THEN
					local.FB.FileOpen.enable := FALSE;
					Status.Error := TRUE;
					Status.ErrorID := local.FB.FileOpen.status;
					local.ErrorStep := local.Step;
					local.Step := vfSTEP_LSF_ERROR;
				END_IF

				// ------------------------------------------------------------------------------------------------------------------------------------------------
				// Wait for incoming command to begin parsing the specified trajectory number.
				// Once parsing is started, commands to process each subsequent trajectory in the same file will start from step vfSTEP_LSF_AWAIT_NEXT_COMMAND.
			vfSTEP_LSF_AWAIT_COMMAND:
				IF (Command.ParseTrajectory) AND NOT (Command.CloseLayer OR Command.AbortLayer OR Command.ResetError) THEN
					IF (Command.OptionalStartingTrajectory > fvp_FIRST_TRAJECTORY_NUMBER) THEN
						local.TrajectoryNumber := Command.OptionalStartingTrajectory;
					ELSE
						local.TrajectoryNumber := fvp_FIRST_TRAJECTORY_NUMBER;
					END_IF
					local.FoundTrajectory := FALSE;
					local.FinalTrajectoryNumber := 0;
					local.FileReadOffset := 0;
					local.Step := vfSTEP_LSF_READ_FILE_DATA;

				ELSIF (Command.CloseLayer) THEN
					local.LayerClosed := TRUE;
					local.Step := vfSTEP_LSF_CLOSE_FILE;

				ELSIF (Command.AbortLayer) THEN
					local.LayerAborted := TRUE;
					local.Step := vfSTEP_LSF_CLOSE_FILE;
				END_IF

				// ------------------------------------------------------------------------------------------------------------------------------------------------
				// Read the next chunk of data large enough to hold the maximum possible trajectory (probably far too long in many cases).
			vfSTEP_LSF_READ_FILE_DATA:
				// Clear the receiving buffer.
				local.StartingByteAddress := ADR(local.DataBuffer);
				brsmemset(local.StartingByteAddress, 0, vfp_LSF_FILE_READ_BUFFER_SIZE);

				// Calculate the number of bytes to read from the file that will include all data for the most complex trajectory.
				local.ReadLengthBytes := (vfp_LSF_NUM_LASERS_PER_SYSTEM * (vfp_LSF_MAX_32BIT_VAL_PER_TRAJ * vfp_LSF_MAX_CHARS_PER_32BIT_VAL)) + vfp_LSF_MAX_CHARS_PER_HEADER;
				// Check that the read buffer size can hold the above.
				IF (local.ReadLengthBytes >= vfp_LSF_FILE_READ_BUFFER_SIZE) THEN
					Status.Error := TRUE;
					Status.ErrorID := vfp_ERR_BUFFER_SIZE;
					local.ErrorStep := local.Step;
					local.Step := vfSTEP_LSF_ERROR;
				ELSE
					// Read the block of data starting at the current FileReadOffset
					local.FB.FileReadEx.ident := local.LocalFileHandle;
					local.FB.FileReadEx.offset := local.FileReadOffset;
					local.FB.FileReadEx.len := local.ReadLengthBytes;
					local.FB.FileReadEx.pDest := local.StartingByteAddress;
					local.FB.FileReadEx.enable := TRUE;
					local.Step := vfSTEP_LSF_WAIT_READ_DONE;
				END_IF

				// ------------------------------------------------------------------------------------------------------------------------------------------------
				// Wait for data read to complete.
			vfSTEP_LSF_WAIT_READ_DONE:
				IF (local.FB.FileReadEx.status = ERR_OK) THEN
					local.FB.FileReadEx.enable := FALSE;
					local.NextByteAddress := local.StartingByteAddress;
					local.TotalBytesRead := local.FB.FileReadEx.bytesread;
					local.CurrentByteIndex := local.NextByteAddress - local.StartingByteAddress;
					IF (local.ParsedHeaderLine) THEN
						local.Step := vfSTEP_LSF_FIND_TRAJECTORY_HDR;
					ELSE
						local.Step := vfSTEP_LSF_PARSE_FILE_HDR;
					END_IF

				ELSIF (local.FB.FileReadEx.status <> ERR_FUB_BUSY) THEN
					local.FB.FileReadEx.enable := FALSE;
					local.TotalBytesRead := 0;
					Status.Error := TRUE;
					Status.ErrorID := local.FB.FileReadEx.status;
					local.ErrorStep := local.Step;
					local.Step := vfSTEP_LSF_CLOSE_FILE;
				END_IF

				// ------------------------------------------------------------------------------------------------------------------------------------------------
				// Parse the file header line.
			vfSTEP_LSF_PARSE_FILE_HDR:

				// TODO: This is a hack - should parse each header element in a separate step to simplify format error identification.
				local.HeaderElement := 0;

				// Read the Build Name.
				local.HeaderElement := local.HeaderElement + 1;
				local.BuildName := '';
				local.CurrentByteIndex := local.NextByteAddress - local.StartingByteAddress;
				local.Status := GetNextString(ADR(local.NextByteAddress), ADR(local.BuildName));

				// Read the Layer Number.
				IF (local.Status = vfp_ERR_OK) THEN
					local.HeaderElement := local.HeaderElement + 1;
					local.ParameterValue := 0;
					local.CurrentByteIndex := local.NextByteAddress - local.StartingByteAddress;
					local.Status := GetNextParameter(ADR(local.NextByteAddress), ADR(local.ParameterValue));
				ELSE
					local.Status := vfp_ERR_BAD_HEADER;
				END_IF

				// Read the Total Number of Layers.
				IF (local.Status = vfp_ERR_OK) THEN
					local.HeaderElement := local.HeaderElement + 1;
					local.ParameterValue := 0;
					local.CurrentByteIndex := local.NextByteAddress - local.StartingByteAddress;
					local.Status := GetNextParameter(ADR(local.NextByteAddress), ADR(local.ParameterValue));
				ELSE
					local.Status := vfp_ERR_BAD_HEADER;
				END_IF

				// Read the Total Number of Trajectories (in this layer).
				IF (local.Status = vfp_ERR_OK) THEN
					local.HeaderElement := local.HeaderElement + 1;
					local.ParameterValue := 0;
					local.CurrentByteIndex := local.NextByteAddress - local.StartingByteAddress;
					local.Status := GetNextParameter(ADR(local.NextByteAddress), ADR(local.ParameterValue));

					IF (local.Status = vfp_ERR_OK) THEN
						IF (local.ParameterValue > 0) THEN
							// The final trajectory number is a multiple of 10.
							local.FinalTrajectoryNumber := LREAL_TO_UINT(local.ParameterValue) * 10;
						ELSE
							local.Status := vfp_ERR_HEADER_INVALID_NUM_TRAJ;
						END_IF
					ELSE
						local.Status := vfp_ERR_BAD_HEADER;
					END_IF
				ELSE
					local.Status := vfp_ERR_BAD_HEADER;
				END_IF

				// Read the Build Plate format.
				IF (local.Status = vfp_ERR_OK) THEN
					local.HeaderElement := local.HeaderElement + 1;
					local.BuildPlateFormat := '';
					local.CurrentByteIndex := local.NextByteAddress - local.StartingByteAddress;
					local.Status := GetNextString(ADR(local.NextByteAddress), ADR(local.BuildPlateFormat));
				ELSE
					local.Status := vfp_ERR_BAD_HEADER;
				END_IF

				IF (local.Status <> vfp_ERR_OK) AND (local.Status <> vfp_ERR_EOL_REACHED) THEN
					Status.Error := TRUE;
					Status.ErrorID := local.Status;
					local.ErrorStep := local.Step;
					local.Step := vfSTEP_LSF_CLOSE_FILE;
				ELSE
					local.CurrentByteIndex := local.NextByteAddress - local.StartingByteAddress;
					local.MaxBytes := local.TotalBytesRead - local.CurrentByteIndex;
					local.Status := FindNextLineStart(ADR(local.NextByteAddress), local.MaxBytes);
					IF (local.Status = vfp_ERR_OK) THEN
						local.ParsedHeaderLine := TRUE;
						local.Step := vfSTEP_LSF_FIND_TRAJECTORY_HDR;
					ELSE
						local.Status := vfp_ERR_MISSING_DATA;
						Status.Error := TRUE;
						Status.ErrorID := local.Status;
						local.ErrorStep := local.Step;
						local.Step := vfSTEP_LSF_CLOSE_FILE;
					END_IF
				END_IF

				// ------------------------------------------------------------------------------------------------------------------------------------------------
				// Find the next trajectory header "Nxxxx" by searching for the next 'N' character without going beyond the end of the buffer.
			vfSTEP_LSF_FIND_TRAJECTORY_HDR:
				local.CurrentByteIndex := local.NextByteAddress - local.StartingByteAddress;
				local.MaxBytes := local.TotalBytesRead - local.CurrentByteIndex;
				local.Status := FindNextTrajectoryStart(ADR(local.NextByteAddress), local.MaxBytes);

				IF (local.Status = vfp_ERR_OK) THEN
					local.Step := vfSTEP_LSF_PARSE_TRAJECTORY_HDR;

				ELSIF (local.Status = vfp_ERR_MISSING_DATA) THEN
					local.FileReadOffset := local.FileReadOffset + (local.NextByteAddress - local.StartingByteAddress);
					local.Step := vfSTEP_LSF_READ_FILE_DATA;

				ELSE
					local.FB.FileReadEx.enable := FALSE;
					local.TotalBytesRead := 0;
					Status.Error := TRUE;
					Status.ErrorID := local.Status;
					local.ErrorStep := local.Step;
					local.Step := vfSTEP_LSF_CLOSE_FILE;
				END_IF

				// ------------------------------------------------------------------------------------------------------------------------------------------------
				// Parse the trajectory header to determine if it matches the desired trajectory number.
				// The trajectory header "Nxxxx" is identical to the G-code line number associated with that trajectory.
				// By convention, the value of xxxx is always 4 digits long, the first trajectory is always N0010, and subsequent trajectories increment by 10.
				// This makes it simple to identify the next "printing" trajectory and allows up to 9 lines of G-code between each.
			vfSTEP_LSF_PARSE_TRAJECTORY_HDR:
				// Read the trajectory identifer "Nxxxx" at the start of the pass.
				local.ParameterValue_string := '';
				local.CurrentByteIndex := local.NextByteAddress - local.StartingByteAddress;
				local.Status := GetNextString(ADR(local.NextByteAddress), ADR(local.ParameterValue_string));

				IF (local.Status = vfp_ERR_OK) THEN

					// Convert the desired trajectory number to a string with the "Nxxxx" format, adding required leading 0s.
					brsitoa(local.TrajectoryNumber, ADR(local.Temp_string));
					IF (local.TrajectoryNumber > 999) THEN
						local.GCodeLineNumber_string := 'N';
					ELSIF (local.TrajectoryNumber > 99) THEN
						local.GCodeLineNumber_string := 'N0';
					ELSIF (local.TrajectoryNumber > 9) THEN
						local.GCodeLineNumber_string := 'N00';
					ELSE
						local.GCodeLineNumber_string := 'N000';
					END_IF
					brsstrcat(ADR(local.GCodeLineNumber_string), ADR(local.Temp_string));

					// Compare the desired trajectory number with that read from the file.
					// If the two match, we have located the desired trajectory, so continue with processing..
					IF (brsstrcmp(ADR(local.GCodeLineNumber_string), ADR(local.ParameterValue_string)) = 0) THEN

						// Identify the trajectory number in the parsed data buffer.
						pParsedData.TrajectoryCircularBuffer[pParsedData.FIFOHeadIndex].TrajectoryNumber := local.TrajectoryNumber;
						local.Step := vfSTEP_LSF_PARSE_NUM_EVENTS;

						// Set the flag indicating that the trajectory marker has been located.
						local.FoundTrajectory := TRUE;
						// Start with the first laser in the trajectory.
						local.LaserNumber := 1;

						// Otherwise, continue searching the file for the desired trajectory number.
					ELSE
						local.FileReadOffset := local.FileReadOffset + (local.NextByteAddress - local.StartingByteAddress);
						local.Step := vfSTEP_LSF_READ_FILE_DATA;
					END_IF

				ELSE
					pParsedData.TrajectoryCircularBuffer[pParsedData.FIFOHeadIndex].ExitCode := local.Status;
					Status.Error := TRUE;
					Status.ErrorID := local.Status;
					local.ErrorStep := local.Step;
					local.Step := vfSTEP_LSF_CLOSE_FILE;
				END_IF

				// ------------------------------------------------------------------------------------------------------------------------------------------------
				// Extract the number of events (laser states) for this trajectory.
			vfSTEP_LSF_PARSE_NUM_EVENTS:
				local.ParameterValue := 0;
				local.CurrentByteIndex := local.NextByteAddress - local.StartingByteAddress;
				local.Status := GetNextParameter(ADR(local.NextByteAddress), ADR(local.ParameterValue));

				IF (local.Status = vfp_ERR_OK) THEN
					IF (local.ParameterValue > 0) THEN
						local.ExpectedNumEvents := LREAL_TO_UINT(local.ParameterValue);
						// Verify that the expected number of events is within the valid range.
						IF (local.ExpectedNumEvents > 0.0) AND (local.ExpectedNumEvents < (vfp_LSF_MAX_32BIT_VAL_PER_TRAJ * 32)) THEN
							local.Step := vfSTEP_LSF_PARSE_LASER_POWERS;
						ELSE
							local.Status := vfp_ERR_INVALID_PARAMETER;
							pParsedData.TrajectoryCircularBuffer[pParsedData.FIFOHeadIndex].ExitCode := local.Status;
							Status.Error := TRUE;
							Status.ErrorID := local.Status;
							local.ErrorStep := local.Step;
							local.Step := vfSTEP_LSF_CLOSE_FILE;
						END_IF
					ELSE
						local.Status := vfp_ERR_INVALID_PARAMETER;
						pParsedData.TrajectoryCircularBuffer[pParsedData.FIFOHeadIndex].ExitCode := local.Status;
						Status.Error := TRUE;
						Status.ErrorID := local.Status;
						local.ErrorStep := local.Step;
						local.Step := vfSTEP_LSF_CLOSE_FILE;
					END_IF

				ELSE
					local.ExpectedNumEvents := 0;
					pParsedData.TrajectoryCircularBuffer[pParsedData.FIFOHeadIndex].ExitCode := local.Status;
					Status.Error := TRUE;
					Status.ErrorID := local.Status;
					local.ErrorStep := local.Step;
					local.Step := vfSTEP_LSF_CLOSE_FILE;
				END_IF

				// ------------------------------------------------------------------------------------------------------------------------------------------------
				// Extract the laser power settings for this trajectory.
			vfSTEP_LSF_PARSE_LASER_POWERS:
				FOR local.LaserPowerValueIndex := 1 TO local.LastLaserNumber DO
					local.ParameterValue := 0;
					local.CurrentByteIndex := local.NextByteAddress - local.StartingByteAddress;
					local.Status := GetNextParameter(ADR(local.NextByteAddress), ADR(local.ParameterValue));

					CASE local.Status OF

						// Interpret the parameter as a LREAL value; more values expected.
						vfp_ERR_OK:
							IF (local.ParameterValue >= 0.0) AND (local.ParameterValue <= 100.0) THEN
								pParsedData.TrajectoryCircularBuffer[pParsedData.FIFOHeadIndex].LaserTrajectoryInfo[local.LaserPowerValueIndex].PowerSetpointPercent := LREAL_TO_REAL(local.ParameterValue);
							ELSE
								local.Status := vfp_ERR_INVALID_PARAMETER;
								pParsedData.TrajectoryCircularBuffer[pParsedData.FIFOHeadIndex].ExitCode := local.Status;
								Status.Error := TRUE;
								Status.ErrorID := local.Status;
								local.ErrorStep := local.Step;
								local.Step := vfSTEP_LSF_CLOSE_FILE;
								EXIT;
							END_IF

							// Interpret the parameter as a REAL value; this is the last laser power value value.
						vfp_ERR_EOL_REACHED:
							IF (local.ParameterValue >= 0.0) AND (local.ParameterValue <= 100.0) THEN
								pParsedData.TrajectoryCircularBuffer[pParsedData.FIFOHeadIndex].LaserTrajectoryInfo[local.LaserPowerValueIndex].PowerSetpointPercent := LREAL_TO_REAL(local.ParameterValue);
							ELSE
								local.Status := vfp_ERR_INVALID_PARAMETER;
								pParsedData.TrajectoryCircularBuffer[pParsedData.FIFOHeadIndex].ExitCode := local.Status;
								Status.Error := TRUE;
								Status.ErrorID := local.Status;
								local.ErrorStep := local.Step;
								local.Step := vfSTEP_LSF_CLOSE_FILE;
								EXIT;
							END_IF

							// Find the start of the next line without going beyond the end of the buffer.
							local.CurrentByteIndex := local.NextByteAddress - local.StartingByteAddress;
							local.MaxBytes := local.TotalBytesRead - local.CurrentByteIndex;
							local.Status := FindNextLineStart(ADR(local.NextByteAddress), local.MaxBytes);
							IF (local.Status = vfp_ERR_OK) THEN
								local.Step := vfSTEP_LSF_PARSE_LASER_STATES;
								EXIT;
							ELSE
								pParsedData.TrajectoryCircularBuffer[pParsedData.FIFOHeadIndex].ExitCode := vfp_ERR_NO_MORE_LINES;
								Status.Error := TRUE;
								Status.ErrorID := local.Status;
								local.ErrorStep := local.Step;
								local.Step := vfSTEP_LSF_CLOSE_FILE;
								EXIT;
							END_IF

							// Found a non-numerical character or encountered end of file (this should not happen while reading laser states).
						ELSE
							pParsedData.TrajectoryCircularBuffer[pParsedData.FIFOHeadIndex].ExitCode := local.Status;
							Status.Error := TRUE;
							Status.ErrorID := local.Status;
							local.ErrorStep := local.Step;
							local.Step := vfSTEP_LSF_CLOSE_FILE;
							EXIT;

					END_CASE
				END_FOR

				// If there were more parameters than the number of lasers, ignore them.
				IF (local.Step = vfSTEP_LSF_PARSE_LASER_POWERS) THEN
					// Find the start of the next line without going beyond the end of the buffer.
					local.CurrentByteIndex := local.NextByteAddress - local.StartingByteAddress;
					local.MaxBytes := local.TotalBytesRead - local.CurrentByteIndex;
					local.Status := FindNextLineStart(ADR(local.NextByteAddress), local.MaxBytes);
					IF (local.Status = vfp_ERR_OK) THEN
						local.Step := vfSTEP_LSF_PARSE_LASER_STATES;
					ELSE
						pParsedData.TrajectoryCircularBuffer[pParsedData.FIFOHeadIndex].ExitCode := vfp_ERR_NO_MORE_LINES;
						Status.Error := TRUE;
						Status.ErrorID := local.Status;
						local.ErrorStep := local.Step;
						local.Step := vfSTEP_LSF_CLOSE_FILE;
					END_IF
				END_IF

				// ------------------------------------------------------------------------------------------------------------------------------------------------
				// Extract all of the 32-bit laser state values for the current laser.
			vfSTEP_LSF_PARSE_LASER_STATES:
				FOR local.LaserStateValueIndex := 1 TO vfp_LSF_MAX_32BIT_VAL_PER_TRAJ DO
					local.ParameterValue := 0;
					local.CurrentByteIndex := local.NextByteAddress - local.StartingByteAddress;
					local.Status := GetNextParameter(ADR(local.NextByteAddress), ADR(local.ParameterValue));

					CASE local.Status OF

						// Interpret the parameter as a UDINT value; more values expected.
						vfp_ERR_OK:
							local.ParameterValue_UDINT := LREAL_TO_UDINT(local.ParameterValue);
							pParsedData.TrajectoryCircularBuffer[pParsedData.FIFOHeadIndex].LaserTrajectoryInfo[local.LaserNumber].StateValue32Bit[local.LaserStateValueIndex] := local.ParameterValue_UDINT;
							pParsedData.TrajectoryCircularBuffer[pParsedData.FIFOHeadIndex].LaserTrajectoryInfo[local.LaserNumber].NumStateValues := local.LaserStateValueIndex;

							// Interpret the parameter as a UDINT value; this is the last value.
						vfp_ERR_EOL_REACHED:
							local.ParameterValue_UDINT := LREAL_TO_UDINT(local.ParameterValue);
							pParsedData.TrajectoryCircularBuffer[pParsedData.FIFOHeadIndex].LaserTrajectoryInfo[local.LaserNumber].StateValue32Bit[local.LaserStateValueIndex] := local.ParameterValue_UDINT;
							pParsedData.TrajectoryCircularBuffer[pParsedData.FIFOHeadIndex].LaserTrajectoryInfo[local.LaserNumber].NumStateValues := local.LaserStateValueIndex;

							// End of line reached, so check that the number of states includes the expected number.
							IF ((local.LaserStateValueIndex * 32) < local.ExpectedNumEvents) OR ((local.LaserStateValueIndex * 32) > (local.ExpectedNumEvents + 32)) THEN
								local.Status := vfp_ERR_WRONG_NUM_STATES;
								pParsedData.TrajectoryCircularBuffer[pParsedData.FIFOHeadIndex].ExitCode := local.Status;
								Status.Error := TRUE;
								Status.ErrorID := local.Status;
								local.ErrorStep := local.Step;
								local.Step := vfSTEP_LSF_CLOSE_FILE;
								EXIT;
							END_IF

							// Find the start of the next line without going beyond the end of the buffer.
							local.CurrentByteIndex := local.NextByteAddress - local.StartingByteAddress;
							local.MaxBytes := local.TotalBytesRead - (local.NextByteAddress - local.StartingByteAddress);
							local.Status := FindNextLineStart(ADR(local.NextByteAddress), local.MaxBytes);
							IF (local.Status = vfp_ERR_OK) THEN
								local.Step := vfSTEP_LSF_SELECT_NEXT_LASER;
								EXIT;
							ELSE
								pParsedData.TrajectoryCircularBuffer[pParsedData.FIFOHeadIndex].ExitCode := vfp_ERR_NO_MORE_LINES;
								Status.Error := TRUE;
								Status.ErrorID := local.Status;
								local.ErrorStep := local.Step;
								local.Step := vfSTEP_LSF_CLOSE_FILE;
								EXIT;
							END_IF

							// Found a non-numerical character or encountered end of file (this should not happen while reading laser states).
						ELSE
							pParsedData.TrajectoryCircularBuffer[pParsedData.FIFOHeadIndex].ExitCode := local.Status;
							Status.Error := TRUE;
							Status.ErrorID := local.Status;
							local.ErrorStep := local.Step;
							local.Step := vfSTEP_LSF_CLOSE_FILE;
							EXIT;

					END_CASE
				END_FOR

				// If there were more than the vfp_LSF_MAX_32BIT_VAL_PER_TRAJ in a trajectory, ignore them and skip to the next laser.
				IF (local.Step = vfSTEP_LSF_PARSE_LASER_STATES) THEN
					// Find the start of the next line without going beyond the end of the buffer.
					local.CurrentByteIndex := local.NextByteAddress - local.StartingByteAddress;
					local.MaxBytes := local.TotalBytesRead - (local.NextByteAddress - local.StartingByteAddress);
					local.Status := FindNextLineStart(ADR(local.NextByteAddress), local.MaxBytes);
					IF (local.Status = vfp_ERR_OK) THEN
						local.Step := vfSTEP_LSF_SELECT_NEXT_LASER;
					ELSE
						pParsedData.TrajectoryCircularBuffer[pParsedData.FIFOHeadIndex].ExitCode := vfp_ERR_NO_MORE_LINES;
						Status.Error := TRUE;
						Status.ErrorID := local.Status;
						local.ErrorStep := local.Step;
						local.Step := vfSTEP_LSF_CLOSE_FILE;
					END_IF
				END_IF

				// ------------------------------------------------------------------------------------------------------------------------------------------------
				// Increment the laser number and continue parsing or indicate that trajectory parsing is complete.
			vfSTEP_LSF_SELECT_NEXT_LASER:
				local.LaserNumber := local.LaserNumber + 1;
				IF (local.LaserNumber <= local.LastLaserNumber) THEN
					local.Step := vfSTEP_LSF_PARSE_LASER_STATES;
				ELSE
					// Notify the caller that the requested trajectory has been parsed.
					Status.ParseTrajectoryComplete := TRUE;
					Status.FinalTrajectoryNumber := local.FinalTrajectoryNumber;
					Status.ParsedTrajectoryNumber := local.TrajectoryNumber;
					local.Step := vfSTEP_LSF_TRAJECTORY_PARSE_DONE;
				END_IF

				// Trajectory parsing is now complete; await command reset.
			vfSTEP_LSF_TRAJECTORY_PARSE_DONE:
				IF (NOT Command.ParseTrajectory) THEN
					Status.ParseTrajectoryComplete := FALSE;
					Status.ParsedTrajectoryNumber := 0;
					local.Step := vfSTEP_LSF_AWAIT_NEXT_COMMAND;
				END_IF

				// ------------------------------------------------------------------------------------------------------------------------------------------------
				// Wait for the next command.
			vfSTEP_LSF_AWAIT_NEXT_COMMAND:
				IF (Command.ParseTrajectory) THEN
					// Increment to the next trajectory number.
					local.FoundTrajectory := FALSE;
					local.TrajectoryNumber := local.TrajectoryNumber + fvp_TRAJECTORY_NUMBER_INCREMENT;
					local.FileReadOffset := local.FileReadOffset + (local.NextByteAddress - local.StartingByteAddress);
					local.Step := vfSTEP_LSF_READ_FILE_DATA;

				ELSIF (Command.CloseLayer) THEN
					local.LayerClosed := TRUE;
					local.Step := vfSTEP_LSF_CLOSE_FILE;

				ELSIF (Command.AbortLayer) THEN
					local.LayerAborted := TRUE;
					local.Step := vfSTEP_LSF_CLOSE_FILE;
				END_IF

				// ------------------------------------------------------------------------------------------------------------------------------------------------
				// Close the file.
			vfSTEP_LSF_CLOSE_FILE:
				local.FB.FileClose.ident := local.LocalFileHandle;
				local.FB.FileClose.enable := TRUE;
				local.Step := vfSTEP_LSF_WAIT_FILE_CLOSED;

				// ------------------------------------------------------------------------------------------------------------------------------------------------
				// Wait for file to complete closing.
			vfSTEP_LSF_WAIT_FILE_CLOSED:
				IF (local.FB.FileClose.status = ERR_OK) THEN
					local.FB.FileClose.enable := FALSE;
					IF (Status.Error) THEN
						local.Step := vfSTEP_LSF_ERROR;
					ELSIF (local.LayerAborted) THEN
						local.Step := vfSTEP_LSF_LAYER_ABORTED;
					ELSE
						local.Step := vfSTEP_LSF_LAYER_CLOSED;
					END_IF

				ELSIF (local.FB.FileClose.status <> ERR_FUB_BUSY) THEN
					local.FB.FileClose.enable := FALSE;
					Status.Error := TRUE;
					Status.ErrorID := local.FB.FileClose.status;
					local.ErrorStep := local.Step;
					local.Step := vfSTEP_LSF_ERROR;
				END_IF

				// ------------------------------------------------------------------------------------------------------------------------------------------------
				// File parsing is now complete.
				// Wait for all commands to be FALSE before returning to IDLE step.
			vfSTEP_LSF_LAYER_CLOSED:
				Status.LayerOpen := FALSE;
				Status.LayerClosed := TRUE;
				local.Step := vfSTEP_LSF_AWAIT_CMD_RESET;

				// ------------------------------------------------------------------------------------------------------------------------------------------------
				// File parsing was aborted.
			vfSTEP_LSF_LAYER_ABORTED:
				Status.LayerOpen := FALSE;
				Status.LayerAborted := TRUE;
				local.Step := vfSTEP_LSF_AWAIT_CMD_RESET;

				// ------------------------------------------------------------------------------------------------------------------------------------------------
				// Jump here on any sort of error and wait for ErrorReset command.
			vfSTEP_LSF_ERROR:
				Status.LayerOpen := FALSE;
				Status.Error := TRUE;
				IF (Command.ResetError) THEN
					Status.Error := FALSE;
					Status.ErrorID := ERR_OK;
					local.Step := vfSTEP_LSF_AWAIT_CMD_RESET;
				END_IF

				// ------------------------------------------------------------------------------------------------------------------------------------------------
				// Wait for all commands to be FALSE before returning to IDLE step.
			vfSTEP_LSF_AWAIT_CMD_RESET:
				IF NOT (Command.ParseTrajectory OR Command.OpenLayer OR Command.CloseLayer OR Command.AbortLayer OR Command.ResetError) THEN
					Status.LayerOpen := FALSE;
					Status.CurrentLayer := 0;
					Status.ParsedTrajectoryNumber := 0;
					Status.ParseTrajectoryComplete := FALSE;
					Status.LayerClosed := FALSE;
					Status.LayerAborted := FALSE;
					Status.Error := FALSE;
					Status.ErrorID := ERR_OK;
					local.Step := vfSTEP_LSF_INITIALIZE;
				END_IF

		END_CASE

	ELSE  // function block NOT enabled

		Active := FALSE;

		Status.LayerOpen := FALSE;
		Status.CurrentLayer := 0;
		Status.ParsedTrajectoryNumber := 0;
		Status.ParseTrajectoryComplete := FALSE;
		Status.LayerClosed := FALSE;
		Status.LayerAborted := FALSE;
		Status.Error := FALSE;
		Status.ErrorID := ERR_OK;

		local.Step := vfSTEP_LSF_INITIALIZE;
		local.ErrorStep := vfSTEP_LSF_INITIALIZE;
		local.FB.FileOpen.enable := FALSE;
		local.FB.FileReadEx.enable := FALSE;
		local.FB.FileClose.enable := FALSE;

	END_IF

	GetSystemErrorText(Status.ErrorID, ADR(Status.ErrorText));

	local.FB.FileOpen();
	local.FB.FileReadEx();
	local.FB.FileClose();

END_FUNCTION_BLOCK
```

#### VfParseFixedEventFile.st - Fixed event file parser
```iecst
FUNCTION_BLOCK VfParseFixedEventFile

	IF (Enable) THEN

		// Trace the currently-active step; the most recent step is in array index [0].
		IF (local.Step <> local.StepTrace[0]) THEN
			// Use the line below to determined the number of scans required for each operation.
			// IF (local.Step <> vfSTEP_FEF_INITIALIZE) AND (local.Step <> vfSTEP_FEF_IDLE) AND (local.Step <> vfSTEP_FEF_AWAIT_NEXT_COMMAND) AND (local.Step <> vfSTEP_FEF_ERROR) AND (local.Step <> vfSTEP_FEF_AWAIT_CMD_RESET) THEN
			FOR local.index := 99 TO 1 BY (-1) DO
				local.StepTrace[local.index] := local.StepTrace[local.index-1];
			END_FOR
			local.StepTrace[0] := local.Step;
		END_IF

		CASE local.Step OF

			// ------------------------------------------------------------------------------------------------------------------------------------------------
			// Initialize parser state.
			vfSTEP_FEF_INITIALIZE:
				Status.LayerFilename_GCode := '';
				Status.LayerFilename_FixedEvents := '';
				Status.LayerOpen := FALSE;
				Status.CurrentLayer := 0;
				Status.ParsedTrajectoryNumber := 0;
				Status.ParseTrajectoryComplete := FALSE;
				Status.LayerClosed := FALSE;
				Status.LayerAborted := FALSE;
				Status.Error := FALSE;
				Status.ErrorID := ERR_OK;

				local.FB.FileOpen.enable := FALSE;
				local.FB.FileReadEx.enable := FALSE;
				local.FB.FileClose.enable := FALSE;

				local.ParsedHeaderLine := FALSE;
				local.FoundTrajectory := FALSE;
				local.TrajectoryNumber := fvp_FIRST_TRAJECTORY_NUMBER;
				local.FinalTrajectoryNumber := 0;
				local.LayerAborted := FALSE;
				local.LayerClosed := FALSE;

				IF NOT (Command.ParseTrajectory OR Command.OpenLayer OR Command.CloseLayer OR Command.AbortLayer OR Command.ResetError) THEN
					local.Step := vfSTEP_FEF_IDLE;
				END_IF

				// ------------------------------------------------------------------------------------------------------------------------------------------------
				// Wait for incoming command to open the specified layer file.
			vfSTEP_FEF_IDLE:
				Active := TRUE;

				Status.LayerFilename_GCode := '';
				Status.LayerFilename_FixedEvents := '';
				local.ParsedHeaderLine := FALSE;
				local.FoundTrajectory := FALSE;
				local.TrajectoryNumber := fvp_FIRST_TRAJECTORY_NUMBER;
				local.FinalTrajectoryNumber := 0;
				local.LayerAborted := FALSE;
				local.LayerClosed := FALSE;

				IF (Command.OpenLayer) AND NOT (Command.CloseLayer OR Command.AbortLayer OR Command.ResetError) THEN
					IF (Command.SelectedBuildLayout > 0) AND (Command.SelectedPrintNumber > 0) THEN
						local.BuildLayout := Command.SelectedBuildLayout;
						local.PrintNumber := Command.SelectedPrintNumber;
						local.LayerNumber := Command.SelectedLayer;
						local.Step := vfSTEP_FEF_CREATE_LAYER_FILENAME;
					END_IF
				ELSIF (Command.AbortLayer) THEN
					local.LayerAborted := TRUE;
					local.Step := vfSTEP_FEF_CLOSE_FILE;
				END_IF

				// ------------------------------------------------------------------------------------------------------------------------------------------------
			vfSTEP_FEF_CREATE_LAYER_FILENAME:

				// Convert the desired build layout number to a string with the "XXXXX" format, adding required leading 0s.
				brsitoa(local.BuildLayout, ADR(local.Temp_string));
				IF (local.BuildLayout > 9999) THEN
					local.BuildLayout_string := '';
				ELSIF (local.BuildLayout > 999) THEN
					local.BuildLayout_string := '0';
				ELSIF (local.BuildLayout > 99) THEN
					local.BuildLayout_string := '00';
				ELSIF (local.BuildLayout > 9) THEN
					local.BuildLayout_string := '000';
				ELSE
					local.BuildLayout_string := '0000';
				END_IF
				brsstrcat(ADR(local.BuildLayout_string), ADR(local.Temp_string));

				// Convert the desired print number to a string with the "YYYY" format, adding required leading 0s.
				brsitoa(local.PrintNumber, ADR(local.Temp_string));
				IF (local.PrintNumber > 999) THEN
					local.PrintNumber_string := '';
				ELSIF (local.PrintNumber > 99) THEN
					local.PrintNumber_string := '0';
				ELSIF (local.PrintNumber > 9) THEN
					local.PrintNumber_string := '00';
				ELSE
					local.PrintNumber_string := '000';
				END_IF
				brsstrcat(ADR(local.PrintNumber_string), ADR(local.Temp_string));

				// Convert the desired layer number to a string with the "nnnnn" format, adding required leading 0s.
				brsitoa(local.LayerNumber, ADR(local.Temp_string));
				IF (local.LayerNumber > 9999) THEN
					local.LayerNumber_string := '';
				ELSIF (local.LayerNumber > 999) THEN
					local.LayerNumber_string := '0';
				ELSIF (local.LayerNumber > 99) THEN
					local.LayerNumber_string := '00';
				ELSIF (local.LayerNumber > 9) THEN
					local.LayerNumber_string := '000';
				ELSE
					local.LayerNumber_string := '0000';
				END_IF
				brsstrcat(ADR(local.LayerNumber_string), ADR(local.Temp_string));

				// Format the complete layer filename.
				// The .vffe file type extension stands for Vulcan Forms Fixed Events
				local.LayerFileName_FixedEvents := 'VF-';
				brsstrcat(ADR(local.LayerFileName_FixedEvents), ADR(local.BuildLayout_string));
				brsstrcat(ADR(local.LayerFileName_FixedEvents), ADR('-'));
				brsstrcat(ADR(local.LayerFileName_FixedEvents), ADR(local.PrintNumber_string));
				brsstrcat(ADR(local.LayerFileName_FixedEvents), ADR('_L'));
				brsstrcat(ADR(local.LayerFileName_FixedEvents), ADR(local.LayerNumber_string));
				brsstrcat(ADR(local.LayerFileName_FixedEvents), ADR('_FixedEvents.vffe'));

				// Format the complete layer filename.
				// The .cnc file type extension stands for a G-code (CNC) motion control file.
				local.LayerFileName_GCode := 'VF-';
				brsstrcat(ADR(local.LayerFileName_GCode), ADR(local.BuildLayout_string));
				brsstrcat(ADR(local.LayerFileName_GCode), ADR('-'));
				brsstrcat(ADR(local.LayerFileName_GCode), ADR(local.PrintNumber_string));
				brsstrcat(ADR(local.LayerFileName_GCode), ADR('_L'));
				brsstrcat(ADR(local.LayerFileName_GCode), ADR(local.LayerNumber_string));
				brsstrcat(ADR(local.LayerFileName_GCode), ADR('_GCode.cnc'));

				Status.LayerFilename_FixedEvents := local.LayerFileName_FixedEvents;
				Status.LayerFilename_GCode := local.LayerFileName_GCode := local.LayerFileName_GCode;
				local.Step := vfSTEP_FEF_OPEN_FILE;

				// ------------------------------------------------------------------------------------------------------------------------------------------------
				// Open the PTR fixed event file for the specified layer in read-only mode.
			vfSTEP_FEF_OPEN_FILE:
				local.FB.FileOpen.pDevice := ADR('CurrentPTRControlFiles');
				local.FB.FileOpen.pFile := ADR(local.LayerFileName_FixedEvents);
				local.FB.FileOpen.mode := fiREAD_ONLY;
				local.FB.FileOpen.enable := TRUE;
				local.Step := vfSTEP_FEF_WAIT_FILE_OPEN;

				// ------------------------------------------------------------------------------------------------------------------------------------------------
				// Wait for file to be open or failure.
			vfSTEP_FEF_WAIT_FILE_OPEN:
				IF (local.FB.FileOpen.status = ERR_OK) THEN
					local.FB.FileOpen.enable := FALSE;
					local.LocalFileHandle := local.FB.FileOpen.ident;
					local.FileReadOffset := 0;
					// Notify the caller that the requested layer is open.
					Status.LayerOpen := TRUE;
					Status.CurrentLayer := local.LayerNumber;
					local.Step := vfSTEP_FEF_AWAIT_COMMAND;

				ELSIF (local.FB.FileOpen.status <> ERR_FUB_BUSY) THEN
					local.FB.FileOpen.enable := FALSE;
					Status.Error := TRUE;
					Status.ErrorID := local.FB.FileOpen.status;
					local.ErrorStep := local.Step;
					local.Step := vfSTEP_FEF_ERROR;
				END_IF

				// ------------------------------------------------------------------------------------------------------------------------------------------------
				// Wait for incoming command to begin parsing the specified trajectory number.
				// Once parsing is started, commands to process each subsequent trajectory in the same file will start from step vfSTEP_FEF_AWAIT_NEXT_COMMAND.
			vfSTEP_FEF_AWAIT_COMMAND:
				IF (Command.ParseTrajectory) AND NOT (Command.CloseLayer OR Command.AbortLayer OR Command.ResetError) THEN
					IF (Command.OptionalStartingTrajectory > fvp_FIRST_TRAJECTORY_NUMBER) THEN
						local.TrajectoryNumber := Command.OptionalStartingTrajectory;
					ELSE
						local.TrajectoryNumber := fvp_FIRST_TRAJECTORY_NUMBER;
					END_IF
					local.FoundTrajectory := FALSE;
					local.FinalTrajectoryNumber := 0;
					local.FileReadOffset := 0;
					local.Step := vfSTEP_FEF_READ_FILE_DATA;

				ELSIF (Command.CloseLayer) THEN
					local.LayerClosed := TRUE;
					local.Step := vfSTEP_FEF_CLOSE_FILE;

				ELSIF (Command.AbortLayer) THEN
					local.LayerAborted := TRUE;
					local.Step := vfSTEP_FEF_CLOSE_FILE;
				END_IF

				// ------------------------------------------------------------------------------------------------------------------------------------------------
				// Read the next chunk of data large enough to contain all of the trajectory parameters.
			vfSTEP_FEF_READ_FILE_DATA:
				// Clear the receiving buffer.
				local.StartingByteAddress := ADR(local.DataBuffer);
				brsmemset(local.StartingByteAddress, 0, vfp_FEF_FILE_READ_BUFFER_SIZE);

				local.ReadLengthBytes := vfp_FEF_FILE_READ_BUFFER_SIZE - 1;

				// Read the block of data starting at the current FileReadOffset.
				local.FB.FileReadEx.ident := local.LocalFileHandle;
				local.FB.FileReadEx.offset := local.FileReadOffset;
				local.FB.FileReadEx.len := local.ReadLengthBytes;
				local.FB.FileReadEx.pDest := local.StartingByteAddress;
				local.FB.FileReadEx.enable := TRUE;
				local.Step := vfSTEP_FEF_WAIT_READ_DONE;

				// ------------------------------------------------------------------------------------------------------------------------------------------------
				// Wait for data read to complete.
			vfSTEP_FEF_WAIT_READ_DONE:
				IF (local.FB.FileReadEx.status = ERR_OK) THEN
					local.FB.FileReadEx.enable := FALSE;
					local.NextByteAddress := local.StartingByteAddress;
					local.TotalBytesRead := local.FB.FileReadEx.bytesread;
					local.CurrentByteIndex := local.NextByteAddress - local.StartingByteAddress;
					IF (local.ParsedHeaderLine) THEN
						local.Step := vfSTEP_FEF_FIND_TRAJECTORY_HDR;
					ELSE
						local.Step := vfSTEP_FEF_PARSE_FILE_HDR;
					END_IF

				ELSIF (local.FB.FileReadEx.status <> ERR_FUB_BUSY) THEN
					local.FB.FileReadEx.enable := FALSE;
					local.TotalBytesRead := 0;
					Status.Error := TRUE;
					Status.ErrorID := local.FB.FileReadEx.status;
					local.ErrorStep := local.Step;
					local.Step := vfSTEP_FEF_CLOSE_FILE;
				END_IF

				// ------------------------------------------------------------------------------------------------------------------------------------------------
				// Parse the file header line.
			vfSTEP_FEF_PARSE_FILE_HDR:

				// TODO: This is a hack - should parse each header element in a separate step to simplify format error identification.
				local.HeaderElement := 0;

				// Read the Build Name.
				local.HeaderElement := local.HeaderElement + 1;
				local.BuildName := '';
				local.CurrentByteIndex := local.NextByteAddress - local.StartingByteAddress;
				local.Status := GetNextString(ADR(local.NextByteAddress), ADR(local.BuildName));

				// Read the Layer Number.
				IF (local.Status = vfp_ERR_OK) THEN
					local.HeaderElement := local.HeaderElement + 1;
					local.ParameterValue := 0;
					local.CurrentByteIndex := local.NextByteAddress - local.StartingByteAddress;
					local.Status := GetNextParameter(ADR(local.NextByteAddress), ADR(local.ParameterValue));
				ELSE
					local.Status := vfp_ERR_BAD_HEADER;
				END_IF

				// Read the Total Number of Layers.
				IF (local.Status = vfp_ERR_OK) THEN
					local.HeaderElement := local.HeaderElement + 1;
					local.ParameterValue := 0;
					local.CurrentByteIndex := local.NextByteAddress - local.StartingByteAddress;
					local.Status := GetNextParameter(ADR(local.NextByteAddress), ADR(local.ParameterValue));
				ELSE
					local.Status := vfp_ERR_BAD_HEADER;
				END_IF

				// Read the Total Number of Trajectories (in this layer).
				IF (local.Status = vfp_ERR_OK) THEN
					local.HeaderElement := local.HeaderElement + 1;
					local.ParameterValue := 0;
					local.CurrentByteIndex := local.NextByteAddress - local.StartingByteAddress;
					local.Status := GetNextParameter(ADR(local.NextByteAddress), ADR(local.ParameterValue));

					IF (local.Status = vfp_ERR_OK) THEN
						IF (local.ParameterValue > 0) THEN
							// The final trajectory number is a multiple of 10.
							local.FinalTrajectoryNumber := LREAL_TO_UINT(local.ParameterValue) * 10;
						ELSE
							local.Status := vfp_ERR_HEADER_INVALID_NUM_TRAJ;
						END_IF
					ELSE
						local.Status := vfp_ERR_BAD_HEADER;
					END_IF
				ELSE
					local.Status := vfp_ERR_BAD_HEADER;
				END_IF

				// Read the Build Plate format.
				IF (local.Status = vfp_ERR_OK) THEN
					local.HeaderElement := local.HeaderElement + 1;
					local.BuildPlateFormat := '';
					local.CurrentByteIndex := local.NextByteAddress - local.StartingByteAddress;
					local.Status := GetNextString(ADR(local.NextByteAddress), ADR(local.BuildPlateFormat));
				ELSE
					local.Status := vfp_ERR_BAD_HEADER;
				END_IF

				IF (local.Status <> vfp_ERR_OK) AND (local.Status <> vfp_ERR_EOL_REACHED) THEN
					Status.Error := TRUE;
					Status.ErrorID := local.Status;
					local.ErrorStep := local.Step;
					local.Step := vfSTEP_FEF_CLOSE_FILE;
				ELSE
					local.CurrentByteIndex := local.NextByteAddress - local.StartingByteAddress;
					local.MaxBytes := local.TotalBytesRead - local.CurrentByteIndex;
					local.Status := FindNextLineStart(ADR(local.NextByteAddress), local.MaxBytes);
					IF (local.Status = vfp_ERR_OK) THEN
						local.ParsedHeaderLine := TRUE;
						local.Step := vfSTEP_FEF_FIND_TRAJECTORY_HDR;
					ELSE
						local.Status := vfp_ERR_MISSING_DATA;
						Status.Error := TRUE;
						Status.ErrorID := local.Status;
						local.ErrorStep := local.Step;
						local.Step := vfSTEP_FEF_CLOSE_FILE;
					END_IF
				END_IF

				// ------------------------------------------------------------------------------------------------------------------------------------------------
				// Find the next trajectory header "Nxxxx" by searching for the next 'N' character without going beyond the end of the buffer.
			vfSTEP_FEF_FIND_TRAJECTORY_HDR:
				local.CurrentByteIndex := local.NextByteAddress - local.StartingByteAddress;
				local.MaxBytes := local.TotalBytesRead - local.CurrentByteIndex;
				local.Status := FindNextTrajectoryStart(ADR(local.NextByteAddress), local.MaxBytes);

				IF (local.Status = vfp_ERR_OK) THEN
					local.Step := vfSTEP_FEF_PARSE_TRAJECTORY_HDR;

				ELSIF (local.Status = vfp_ERR_MISSING_DATA) THEN
					local.FileReadOffset := local.FileReadOffset + (local.NextByteAddress - local.StartingByteAddress);
					local.Step := vfSTEP_FEF_READ_FILE_DATA;

				ELSE
					local.FB.FileReadEx.enable := FALSE;
					local.TotalBytesRead := 0;
					Status.Error := TRUE;
					Status.ErrorID := local.Status;
					local.ErrorStep := local.Step;
					local.Step := vfSTEP_FEF_CLOSE_FILE;
				END_IF

				// ------------------------------------------------------------------------------------------------------------------------------------------------
				// Parse the trajectory header to determine if it matches the desired trajectory number.
				// The trajectory header "Nxxxx" is identical to the G-code line number associated with that trajectory.
				// By convention, the value of xxxx is always 4 digits long, the first trajectory is always N0010, and subsequent trajectories increment by 10.
				// This makes it simple to identify the next "printing" trajectory and allows up to 9 lines of G-code between each.
			vfSTEP_FEF_PARSE_TRAJECTORY_HDR:
				// Read the trajectory identifer "Nxxxx" at the start of the pass.
				local.ParameterValue_string := '';
				local.CurrentByteIndex := local.NextByteAddress - local.StartingByteAddress;
				local.Status := GetNextString(ADR(local.NextByteAddress), ADR(local.ParameterValue_string));

				IF (local.Status = vfp_ERR_OK) THEN

					// Convert the desired trajectory number to a string with the "Nxxxx" format, adding required leading 0s.
					brsitoa(local.TrajectoryNumber, ADR(local.Temp_string));
					IF (local.TrajectoryNumber > 999) THEN
						local.GCodeLineNumber_string := 'N';
					ELSIF (local.TrajectoryNumber > 99) THEN
						local.GCodeLineNumber_string := 'N0';
					ELSIF (local.TrajectoryNumber > 9) THEN
						local.GCodeLineNumber_string := 'N00';
					ELSE
						local.GCodeLineNumber_string := 'N000';
					END_IF
					brsstrcat(ADR(local.GCodeLineNumber_string), ADR(local.Temp_string));

					// Compare the desired trajectory number with that read from the file.
					// If the two match, we have located the desired trajectory, so continue with processing..
					IF (brsstrcmp(ADR(local.GCodeLineNumber_string), ADR(local.ParameterValue_string)) = 0) THEN

						// Identify the trajectory number in the parsed data buffer.
						pParsedData.TrajectoryCircularBuffer[pParsedData.FIFOHeadIndex].TrajectoryNumber := local.TrajectoryNumber;
						local.Step := vfSTEP_FEF_PARSE_MASTER_AXIS;

						// Set the flag indicating that the trajectory marker has been located.
						local.FoundTrajectory := TRUE;

						// Otherwise, continue searching the file for the desired trajectory number.
					ELSE
						local.FileReadOffset := local.FileReadOffset + (local.NextByteAddress - local.StartingByteAddress);
						local.Step := vfSTEP_FEF_READ_FILE_DATA;
					END_IF

				ELSE
					pParsedData.TrajectoryCircularBuffer[pParsedData.FIFOHeadIndex].ExitCode := local.Status;
					Status.Error := TRUE;
					Status.ErrorID := local.Status;
					local.ErrorStep := local.Step;
					local.Step := vfSTEP_FEF_CLOSE_FILE;
				END_IF

				// ------------------------------------------------------------------------------------------------------------------------------------------------
				// Extract the master axis (X or Y) for this trajectory.
			vfSTEP_FEF_PARSE_MASTER_AXIS:
				local.ParameterValue_string := '';
				local.CurrentByteIndex := local.NextByteAddress - local.StartingByteAddress;
				local.Status := GetNextString(ADR(local.NextByteAddress), ADR(local.ParameterValue_string));

				IF (local.Status = vfp_ERR_OK) THEN

					IF (brsstrcmp(ADR('X'), ADR(local.ParameterValue_string)) = 0) THEN
						local.MasterAxis := vfp_FEF_MASTER_AXIS_X;
						pParsedData.TrajectoryCircularBuffer[pParsedData.FIFOHeadIndex].MasterAxis := local.MasterAxis;
						local.Step := vfSTEP_FEF_PARSE_START_POSN;
					ELSIF (brsstrcmp(ADR('Y'), ADR(local.ParameterValue_string)) = 0) THEN
						local.MasterAxis := vfp_FEF_MASTER_AXIS_Y;
						pParsedData.TrajectoryCircularBuffer[pParsedData.FIFOHeadIndex].MasterAxis := local.MasterAxis;
						local.Step := vfSTEP_FEF_PARSE_START_POSN;
					ELSE
						local.Status := vfp_ERR_INVALID_PARAMETER;
						pParsedData.TrajectoryCircularBuffer[pParsedData.FIFOHeadIndex].ExitCode := local.Status;
						Status.Error := TRUE;
						Status.ErrorID := local.Status;
						local.ErrorStep := local.Step;
						local.Step := vfSTEP_FEF_CLOSE_FILE;
					END_IF

				ELSE
					pParsedData.TrajectoryCircularBuffer[pParsedData.FIFOHeadIndex].ExitCode := local.Status;
					Status.Error := TRUE;
					Status.ErrorID := local.Status;
					local.ErrorStep := local.Step;
					local.Step := vfSTEP_FEF_CLOSE_FILE;
				END_IF

				// ------------------------------------------------------------------------------------------------------------------------------------------------
				// Extract the start position for this trajectory.
			vfSTEP_FEF_PARSE_START_POSN:
				local.ParameterValue := 0;
				local.CurrentByteIndex := local.NextByteAddress - local.StartingByteAddress;
				local.Status := GetNextParameter(ADR(local.NextByteAddress), ADR(local.ParameterValue));

				IF (local.Status = vfp_ERR_OK) THEN

					// Interpret the parameter as a LREAL value.
					IF (local.ParameterValue > 0.0) AND (local.ParameterValue < vfp_FEF_MAX_X_Y_POSN_MM) THEN
						local.StartPosition := LREAL_TO_REAL(local.ParameterValue);
						pParsedData.TrajectoryCircularBuffer[pParsedData.FIFOHeadIndex].StartPositionMM := local.StartPosition;
						local.Step := vfSTEP_FEF_PARSE_END_POSN;
					ELSE
						local.Status := vfp_ERR_INVALID_PARAMETER;
						pParsedData.TrajectoryCircularBuffer[pParsedData.FIFOHeadIndex].ExitCode := local.Status;
						Status.Error := TRUE;
						Status.ErrorID := local.Status;
						local.ErrorStep := local.Step;
						local.Step := vfSTEP_FEF_CLOSE_FILE;
					END_IF

				ELSE
					pParsedData.TrajectoryCircularBuffer[pParsedData.FIFOHeadIndex].ExitCode := local.Status;
					Status.Error := TRUE;
					Status.ErrorID := local.Status;
					local.ErrorStep := local.Step;
					local.Step := vfSTEP_FEF_CLOSE_FILE;
				END_IF

				// ------------------------------------------------------------------------------------------------------------------------------------------------
				// Extract the end position for this trajectory.
			vfSTEP_FEF_PARSE_END_POSN:
				local.ParameterValue := 0;
				local.CurrentByteIndex := local.NextByteAddress - local.StartingByteAddress;
				local.Status := GetNextParameter(ADR(local.NextByteAddress), ADR(local.ParameterValue));

				IF (local.Status = vfp_ERR_OK) THEN

					// Interpret the parameter as a LREAL value.
					IF (local.ParameterValue > 0.0) AND (local.ParameterValue < vfp_FEF_MAX_X_Y_POSN_MM) AND (local.ParameterValue > REAL_TO_LREAL(local.StartPosition)) THEN
						local.EndPosition := LREAL_TO_REAL(local.ParameterValue);
						pParsedData.TrajectoryCircularBuffer[pParsedData.FIFOHeadIndex].EndPositionMM := local.EndPosition;
						local.Step := vfSTEP_FEF_PARSE_EVENT_PERIOD;
					ELSE
						local.Status := vfp_ERR_INVALID_PARAMETER;
						pParsedData.TrajectoryCircularBuffer[pParsedData.FIFOHeadIndex].ExitCode := local.Status;
						Status.Error := TRUE;
						Status.ErrorID := local.Status;
						local.ErrorStep := local.Step;
						local.Step := vfSTEP_FEF_CLOSE_FILE;
					END_IF

				ELSE
					pParsedData.TrajectoryCircularBuffer[pParsedData.FIFOHeadIndex].ExitCode := local.Status;
					Status.Error := TRUE;
					Status.ErrorID := local.Status;
					local.ErrorStep := local.Step;
					local.Step := vfSTEP_FEF_CLOSE_FILE;
				END_IF

				// ------------------------------------------------------------------------------------------------------------------------------------------------
				// Extract the event period for this trajectory.
			vfSTEP_FEF_PARSE_EVENT_PERIOD:
				local.ParameterValue := 0;
				local.CurrentByteIndex := local.NextByteAddress - local.StartingByteAddress;
				local.Status := GetNextParameter(ADR(local.NextByteAddress), ADR(local.ParameterValue));

				// This is the last parameter on the line, so EOL_REACHED is expected.
				IF (local.Status = vfp_ERR_OK) OR (local.Status = vfp_ERR_EOL_REACHED) THEN

					// Interpret the parameter as a LREAL value.
					IF (local.ParameterValue > 0.0) AND (local.ParameterValue < 1.0) THEN
						local.EventPeriod := LREAL_TO_REAL(local.ParameterValue);
						pParsedData.TrajectoryCircularBuffer[pParsedData.FIFOHeadIndex].EventPeriodMM := local.EventPeriod;

						Status.ParseTrajectoryComplete := TRUE;
						Status.FinalTrajectoryNumber := local.FinalTrajectoryNumber;
						Status.ParsedTrajectoryNumber := local.TrajectoryNumber;
						local.Step := vfSTEP_FEF_TRAJECTORY_PARSE_DONE;
					ELSE
						local.Status := vfp_ERR_INVALID_PARAMETER;
						pParsedData.TrajectoryCircularBuffer[pParsedData.FIFOHeadIndex].ExitCode := local.Status;
						Status.Error := TRUE;
						Status.ErrorID := local.Status;
						local.ErrorStep := local.Step;
						local.Step := vfSTEP_FEF_CLOSE_FILE;
					END_IF

				ELSE
					pParsedData.TrajectoryCircularBuffer[pParsedData.FIFOHeadIndex].ExitCode := local.Status;
					Status.Error := TRUE;
					Status.ErrorID := local.Status;
					local.ErrorStep := local.Step;
					local.Step := vfSTEP_FEF_CLOSE_FILE;
				END_IF

				// ------------------------------------------------------------------------------------------------------------------------------------------------
				// Trajectory parsing is now complete; await command reset.
			vfSTEP_FEF_TRAJECTORY_PARSE_DONE:
				IF (NOT Command.ParseTrajectory) THEN
					Status.ParseTrajectoryComplete := FALSE;
					Status.ParsedTrajectoryNumber := 0;
					local.Step := vfSTEP_FEF_AWAIT_NEXT_COMMAND;
				END_IF

				// ------------------------------------------------------------------------------------------------------------------------------------------------
				// Wait for the next command.
			vfSTEP_FEF_AWAIT_NEXT_COMMAND:
				IF (Command.ParseTrajectory) THEN
					// Increment to the next trajectory number.
					local.FoundTrajectory := FALSE;
					local.TrajectoryNumber := local.TrajectoryNumber + fvp_TRAJECTORY_NUMBER_INCREMENT;
					local.FileReadOffset := local.FileReadOffset + (local.NextByteAddress - local.StartingByteAddress);
					local.Step := vfSTEP_FEF_READ_FILE_DATA;

				ELSIF (Command.CloseLayer) THEN
					local.LayerClosed := TRUE;
					local.Step := vfSTEP_FEF_CLOSE_FILE;

				ELSIF (Command.AbortLayer) THEN
					local.LayerAborted := TRUE;
					local.Step := vfSTEP_FEF_CLOSE_FILE;
				END_IF

				// ------------------------------------------------------------------------------------------------------------------------------------------------
				// Close the file.
			vfSTEP_FEF_CLOSE_FILE:
				local.FB.FileClose.ident := local.LocalFileHandle;
				local.FB.FileClose.enable := TRUE;
				local.Step := vfSTEP_FEF_WAIT_FILE_CLOSED;

				// ------------------------------------------------------------------------------------------------------------------------------------------------
				// Wait for file to complete closing.
			vfSTEP_FEF_WAIT_FILE_CLOSED:
				IF (local.FB.FileClose.status = ERR_OK) THEN
					local.FB.FileClose.enable := FALSE;
					IF (Status.Error) THEN
						local.Step := vfSTEP_FEF_ERROR;
					ELSIF (local.LayerAborted) THEN
						local.Step := vfSTEP_FEF_LAYER_ABORTED;
					ELSE
						local.Step := vfSTEP_FEF_LAYER_CLOSED;
					END_IF

				ELSIF (local.FB.FileClose.status <> ERR_FUB_BUSY) THEN
					local.FB.FileClose.enable := FALSE;
					Status.Error := TRUE;
					Status.ErrorID := local.FB.FileClose.status;
					local.ErrorStep := local.Step;
					local.Step := vfSTEP_FEF_ERROR;
				END_IF

				// ------------------------------------------------------------------------------------------------------------------------------------------------
				// File parsing is now complete.
				// Wait for all commands to be FALSE before returning to IDLE step.
			vfSTEP_FEF_LAYER_CLOSED:
				Status.LayerOpen := FALSE;
				Status.LayerClosed := TRUE;
				local.Step := vfSTEP_FEF_AWAIT_CMD_RESET;

				// ------------------------------------------------------------------------------------------------------------------------------------------------
				// File parsing was aborted.
			vfSTEP_FEF_LAYER_ABORTED:
				Status.LayerOpen := FALSE;
				Status.LayerAborted := TRUE;
				local.Step := vfSTEP_FEF_AWAIT_CMD_RESET;

				// ------------------------------------------------------------------------------------------------------------------------------------------------
				// Jump here on any sort of error and wait for ErrorReset command.
			vfSTEP_FEF_ERROR:
				Status.LayerOpen := FALSE;
				Status.Error := TRUE;
				IF (Command.ResetError) THEN
					Status.Error := FALSE;
					Status.ErrorID := ERR_OK;
					local.Step := vfSTEP_FEF_AWAIT_CMD_RESET;
				END_IF

				// ------------------------------------------------------------------------------------------------------------------------------------------------
				// Wait for all commands to be FALSE before returning to IDLE step.
			vfSTEP_FEF_AWAIT_CMD_RESET:
				IF NOT (Command.ParseTrajectory OR Command.OpenLayer OR Command.CloseLayer OR Command.AbortLayer OR Command.ResetError) THEN
					Status.LayerOpen := FALSE;
					Status.CurrentLayer := 0;
					Status.ParsedTrajectoryNumber := 0;
					Status.ParseTrajectoryComplete := FALSE;
					Status.LayerClosed := FALSE;
					Status.LayerAborted := FALSE;
					Status.Error := FALSE;
					Status.ErrorID := ERR_OK;
					local.Step := vfSTEP_FEF_INITIALIZE;
				END_IF

		END_CASE

	ELSE  // function block NOT enabled

		Active := FALSE;

		Status.LayerOpen := FALSE;
		Status.CurrentLayer := 0;
		Status.ParsedTrajectoryNumber := 0;
		Status.ParseTrajectoryComplete := FALSE;
		Status.LayerClosed := FALSE;
		Status.LayerAborted := FALSE;
		Status.Error := FALSE;
		Status.ErrorID := ERR_OK;

		local.Step := vfSTEP_FEF_INITIALIZE;
		local.ErrorStep := vfSTEP_FEF_INITIALIZE;
		local.FB.FileOpen.enable := FALSE;
		local.FB.FileReadEx.enable := FALSE;
		local.FB.FileClose.enable := FALSE;

	END_IF

	GetSystemErrorText(Status.ErrorID, ADR(Status.ErrorText));

	local.FB.FileOpen();
	local.FB.FileReadEx();
	local.FB.FileClose();

END_FUNCTION_BLOCK
```

#### VfSMRConnect.st - not currently in use
```iecst
FUNCTION_BLOCK VfSMRConnect

	IF (Execute) THEN

		// Trace the currently-active step; the most recent step is in array index [0].
		IF (Internal.Step <> Internal.StepTrace[0]) THEN
			FOR Internal.index := 99 TO 1 BY (-1) DO
				Internal.StepTrace[Internal.index] := Internal.StepTrace[Internal.index-1];
			END_FOR
			Internal.StepTrace[0] := Internal.Step;
		END_IF;

		// Main state machine
		CASE Internal.Step OF

			// Waiting for Execute
			vfSMR_CNCT_STEP_IDLE:
				Internal.Step := vfSMR_CNCT_STEP_CONNECT_SMR1;

			// Establish connection to local media where target file will be placed
			vfSMR_CNCT_STEP_CONNECT_SMR1:
				Internal.FB.DevLinkLocalSMR.pDevice := pLocalSMRDriveName;
				Internal.FB.DevLinkLocalSMR.pParam := pLocalSMRDrive;
				Internal.FB.DevLinkLocalSMR.enable := TRUE;
				Internal.Step := vfSMR_CNCT_STEP_CONNECT_SMR2;

			// Wait for successful connection
			vfSMR_CNCT_STEP_CONNECT_SMR2:
				IF (Internal.FB.DevLinkLocalSMR.status = ERR_OK) THEN
					Internal.FB.DevLinkLocalSMR.enable := FALSE;
					LocalSMRDriveHandle := Internal.FB.DevLinkLocalSMR.handle;
					Internal.Step := vfSMR_CNCT_STEP_CONNECT_PTR1;

				ELSIF (Internal.FB.DevLinkLocalSMR.status <> ERR_FUB_BUSY) THEN
					Internal.FB.DevLinkLocalSMR.enable := FALSE;
					Internal.ErrorStep := Internal.Step;
					Error := TRUE;
					ErrorID := Internal.FB.DevLinkLocalSMR.status;
					Internal.Step := vfSMR_CNCT_STEP_DISCONNECT1;

				END_IF

			// Establish connection to local media where target file will be placed
			vfSMR_CNCT_STEP_CONNECT_PTR1:
				Internal.FB.DevLinkLocalPTR.pDevice := pLocalPTRDriveName;
				Internal.FB.DevLinkLocalPTR.pParam := pLocalPTRDrive;
				Internal.FB.DevLinkLocalPTR.enable := TRUE;
				Internal.Step := vfSMR_CNCT_STEP_CONNECT_PTR2;

			// Wait for successful connection
			vfSMR_CNCT_STEP_CONNECT_PTR2:
				IF (Internal.FB.DevLinkLocalPTR.status = ERR_OK) THEN
					Internal.FB.DevLinkLocalPTR.enable := FALSE;
					LocalPTRDriveHandle := Internal.FB.DevLinkLocalPTR.handle;
					Internal.Step := vfSMR_CNCT_STEP_CONNECT_LCR1;

				ELSIF (Internal.FB.DevLinkLocalPTR.status <> ERR_FUB_BUSY) THEN
					Internal.FB.DevLinkLocalPTR.enable := FALSE;
					Internal.ErrorStep := Internal.Step;
					Error := TRUE;
					ErrorID := Internal.FB.DevLinkLocalPTR.status;
					Internal.Step := vfSMR_CNCT_STEP_DISCONNECT1;

				END_IF

			// Establish connection to local media where target file will be placed
			vfSMR_CNCT_STEP_CONNECT_LCR1:
				Internal.FB.DevLinkLocalLCR.pDevice := pLocalLCRDriveName;
				Internal.FB.DevLinkLocalLCR.pParam := pLocalLCRDrive;
				Internal.FB.DevLinkLocalLCR.enable := TRUE;
				Internal.Step := vfSMR_CNCT_STEP_CONNECT_LCR2;

			// Wait for successful connection
			vfSMR_CNCT_STEP_CONNECT_LCR2:
				IF (Internal.FB.DevLinkLocalLCR.status = ERR_OK) THEN
					Internal.FB.DevLinkLocalLCR.enable := FALSE;
					LocalLCRDriveHandle := Internal.FB.DevLinkLocalLCR.handle;
					Internal.Step := vfSMR_CNCT_STEP_CONNECT_REMOTE1;

				ELSIF (Internal.FB.DevLinkLocalLCR.status <> ERR_FUB_BUSY) THEN
					Internal.FB.DevLinkLocalLCR.enable := FALSE;
					Internal.ErrorStep := Internal.Step;
					Error := TRUE;
					ErrorID := Internal.FB.DevLinkLocalLCR.status;
					Internal.Step := vfSMR_CNCT_STEP_DISCONNECT1;

				END_IF

			// Establish connection to remote media where target file resides
			vfSMR_CNCT_STEP_CONNECT_REMOTE1:
				Internal.FB.DevLinkRemote.pDevice := pRemoteDriveName;
				Internal.FB.DevLinkRemote.pParam := pRemoteDrive;
				Internal.FB.DevLinkRemote.enable := TRUE;
				Internal.Step := vfSMR_CNCT_STEP_CONNECT_REMOTE2;

			// Wait for successful connection
			vfSMR_CNCT_STEP_CONNECT_REMOTE2:
				IF (Internal.FB.DevLinkRemote.status = ERR_OK) THEN
					Internal.FB.DevLinkRemote.enable := FALSE;
					RemoteDriveHandle := Internal.FB.DevLinkRemote.handle;
					Internal.Step := vfSMR_CNCT_STEP_DONE;

				ELSIF (Internal.FB.DevLinkRemote.status <> ERR_FUB_BUSY) THEN
					Internal.FB.DevLinkRemote.enable := FALSE;
					Internal.ErrorStep := Internal.Step;
					Error := TRUE;
					ErrorID := Internal.FB.DevLinkRemote.status;
					Internal.Step := vfSMR_CNCT_STEP_DISCONNECT1;

				END_IF

			// Wait for incoming command
			vfSMR_CNCT_STEP_DONE:
				Done := TRUE;

			// Disconnect from all media
			vfSMR_CNCT_STEP_DISCONNECT1:
				IF (LocalSMRDriveHandle <> 0) THEN
					Internal.FB.DevUnlinkLocalSMR.handle := LocalSMRDriveHandle;
					Internal.FB.DevUnlinkLocalSMR.enable := TRUE;
				END_IF
				IF (LocalPTRDriveHandle <> 0) THEN
					Internal.FB.DevUnlinkLocalPTR.handle := LocalPTRDriveHandle;
					Internal.FB.DevUnlinkLocalPTR.enable := TRUE;
				END_IF
				IF (RemoteDriveHandle <> 0) THEN
					Internal.FB.DevUnlinkRemote.handle := RemoteDriveHandle;
					Internal.FB.DevUnlinkRemote.enable := TRUE;
				END_IF
				Internal.Step := vfSMR_CNCT_STEP_DISCONNECT2;

			vfSMR_CNCT_STEP_DISCONNECT2:
				// Wait for confirmation that both devices are unlinked
				IF (((Internal.FB.DevUnlinkLocalSMR.status = ERR_OK) OR (NOT Internal.FB.DevUnlinkLocalSMR.enable)) AND
					((Internal.FB.DevUnlinkLocalPTR.status = ERR_OK) OR (NOT Internal.FB.DevUnlinkLocalPTR.enable)) AND
					((Internal.FB.DevUnlinkRemote.status = ERR_OK) OR (NOT Internal.FB.DevUnlinkRemote.enable))) THEN
					LocalSMRDriveHandle := 0;
					LocalPTRDriveHandle := 0;
					RemoteDriveHandle := 0;
					Internal.Step := vfSMR_CNCT_STEP_ERROR;
				END_IF

			vfSMR_CNCT_STEP_ERROR:

				IF (ErrorReset) THEN
					Internal.Step := vfSMR_CNCT_STEP_ERROR_RESET;
				END_IF

			vfSMR_CNCT_STEP_ERROR_RESET:

		END_CASE

	ELSE // NOT Execute
		Internal.Step := vfSMR_CNCT_STEP_IDLE;
		Done := FALSE;
		Error := FALSE;
		ErrorID := ERR_OK;
		Internal.FB.DevLinkLocalSMR.enable := FALSE;
		Internal.FB.DevLinkLocalPTR.enable := FALSE;
		Internal.FB.DevLinkRemote.enable := FALSE;
		Internal.FB.DevUnlinkLocalSMR.enable := FALSE;
		Internal.FB.DevUnlinkLocalPTR.enable := FALSE;
		Internal.FB.DevUnlinkRemote.enable := FALSE;

	END_IF

	// Calling all FBs
	Internal.FB.DevLinkLocalSMR();
	Internal.FB.DevLinkLocalPTR();
	Internal.FB.DevLinkLocalLCR();
	Internal.FB.DevLinkRemote();

	Internal.FB.DevUnlinkLocalSMR();
	Internal.FB.DevUnlinkLocalPTR();
	Internal.FB.DevUnlinkRemote();
	Internal.FB.DevUnlinkLocalLCR();

END_FUNCTION_BLOCK
```
